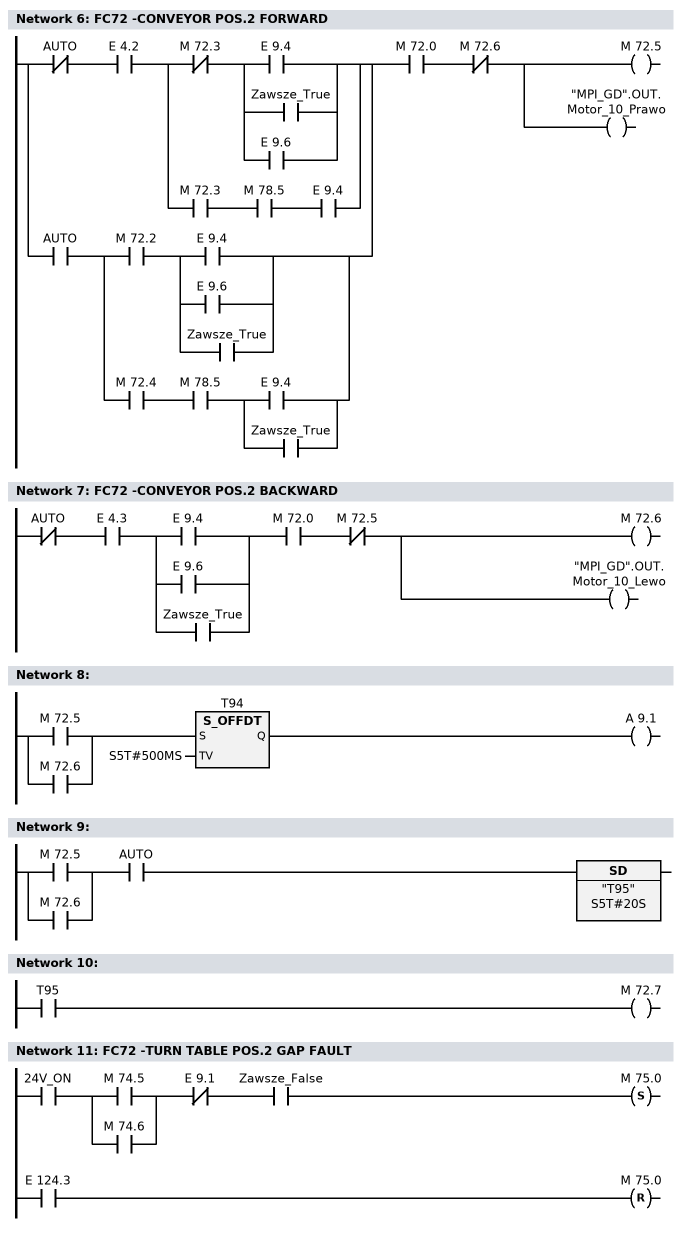
[picture p72: CONV_2 networks 6-11]
NETWORK
TITLE = FC72 -CONVEYOR POS.2 FORWARD
//Q8.2. Przenosnik jedzie do przodu
      A(;
      AN    "AUTO";
      A     "E 4.2";
      A(;
      AN    "M 72.3";
      A(;
      O     "E 9.4";
      O     "Zawsze_True";
      O     "E 9.6";
      );
      O;
      A     "M 72.3";
      A     "M 78.5";
      A     "E 9.4";
      );
      O;
      A     "AUTO";
      A(;
      A     "M 72.2";
      A(;
      O     "E 9.4";
      O     "E 9.6";
      O     "Zawsze_True";
      );
      O;
      A     "M 72.4";
      A     "M 78.5";
      A(;
      O     "E 9.4";
      O     "Zawsze_True";
      );
      );
      );
      A     "M 72.0";
      AN    "M 72.6";
      =     "M 72.5";
      =     "MPI_GD".OUT.Motor_10_Prawo;
NETWORK
TITLE = FC72 -CONVEYOR POS.2 BACKWARD
//Q8.3 przenosnik jedzie do tylu
      AN    "AUTO";
      A     "E 4.3";
      A(;
      O     "E 9.4";
      O     "E 9.6";
      O     "Zawsze_True";
      );
      A     "M 72.0";
      AN    "M 72.5";
      =     "M 72.6";
      =     "MPI_GD".OUT.Motor_10_Lewo;
NETWORK
TITLE =
      A(;
      O     "M 72.5";
      O     "M 72.6";
      );
      L     S5T#500MS;
      SF    "T94";
      NOP   0;
      NOP   0;
      NOP   0;
      A     "T94";
      =     "A 9.1";
NETWORK
TITLE =
      A(;
      O     "M 72.5";
      O     "M 72.6";
      );
      A     "AUTO";
      L     S5T#20S;
      SD    "T95";
NETWORK
TITLE =
      A     "T95";
      =     "M 72.7";
NETWORK
TITLE = FC72 -TURN TABLE POS.2 GAP FAULT
//Zablokowane
      A     "24V_ON";
      A(;
      O     "M 74.5";
      O     "M 74.6";
      );
      AN    "E 9.1";
      A     "Zawsze_False";
      S     "M 75.0";
      A     "E 124.3";
      R     "M 75.0";
      NOP   0;
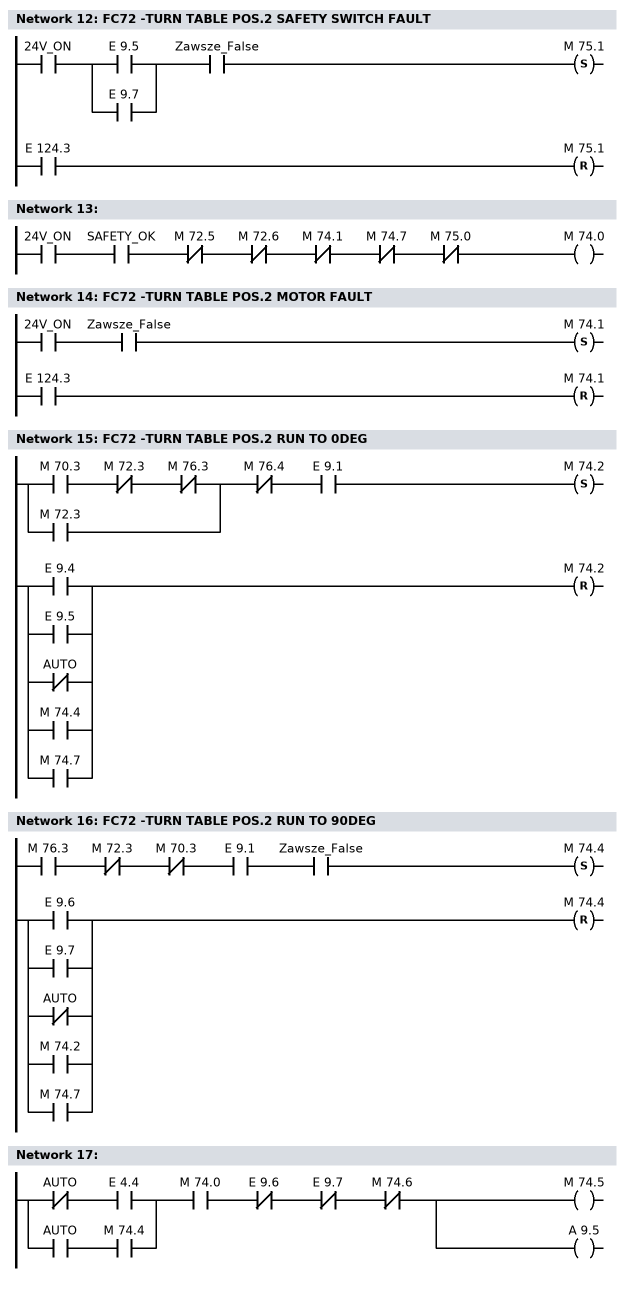
NETWORK
TITLE = FC72 -TURN TABLE POS.2 SAFETY SWITCH FAULT
//Zablokowane
      A     "24V_ON";
      A(;
      O     "E 9.5";
      O     "E 9.7";
      );
      A     "Zawsze_False";
      S     "M 75.1";
      A     "E 124.3";
      R     "M 75.1";
      NOP   0;
NETWORK
TITLE =
      A     "24V_ON";
      A     "SAFETY_OK";
      AN    "M 72.5";
      AN    "M 72.6";
      AN    "M 74.1";
      AN    "M 74.7";
      AN    "M 75.0";
      =     "M 74.0";
NETWORK
TITLE = FC72 -TURN TABLE POS.2 MOTOR FAULT
//Zablokowane.Silnik obrotnica
      A     "24V_ON";
      A     "Zawsze_False";
      S     "M 74.1";
      A     "E 124.3";
      R     "M 74.1";
      NOP   0;
NETWORK
TITLE = FC72 -TURN TABLE POS.2 RUN TO 0DEG
      A(;
      A     "M 70.3";
      AN    "M 72.3";
      AN    "M 76.3";
      O     "M 72.3";
      );
      AN    "M 76.4";
      A     "E 9.1";
      S     "M 74.2";
      A(;
      O     "E 9.4";
      O     "E 9.5";
      ON    "AUTO";
      O     "M 74.4";
      O     "M 74.7";
      );
      R     "M 74.2";
      NOP   0;
NETWORK
TITLE = FC72 -TURN TABLE POS.2 RUN TO 90DEG
//Zablokowane
      A     "M 76.3";
      AN    "M 72.3";
      AN    "M 70.3";
      A     "E 9.1";
      A     "Zawsze_False";
      S     "M 74.4";
      A(;
      O     "E 9.6";
      O     "E 9.7";
      ON    "AUTO";
      O     "M 74.2";
      O     "M 74.7";
      );
      R     "M 74.4";
      NOP   0;
NETWORK
TITLE =
      A(;
      AN    "AUTO";
      A     "E 4.4";
      O;
      A     "AUTO";
      A     "M 74.4";
      );
      A     "M 74.0";
      AN    "E 9.6";
      AN    "E 9.7";
      AN    "M 74.6";
      =     "M 74.5";
      =     "A 9.5";
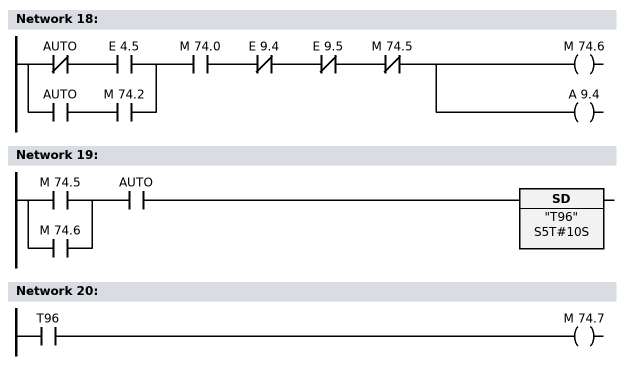
NETWORK
TITLE =
      A(;
      AN    "AUTO";
      A     "E 4.5";
      O;
      A     "AUTO";
      A     "M 74.2";
      );
      A     "M 74.0";
      AN    "E 9.4";
      AN    "E 9.5";
      AN    "M 74.5";
      =     "M 74.6";
      =     "A 9.4";
NETWORK
TITLE =
      A(;
      O     "M 74.5";
      O     "M 74.6";
      );
      A     "AUTO";
      L     S5T#10S;
      SD    "T96";
NETWORK
TITLE =
      A     "T96";
      =     "M 74.7";
END_FUNCTION

FUNCTION "Komunikacja_GD" : VOID	// FC 100
VERSION : 0.1
BEGIN
NETWORK
TITLE =
//Ten network celowo jest wolny
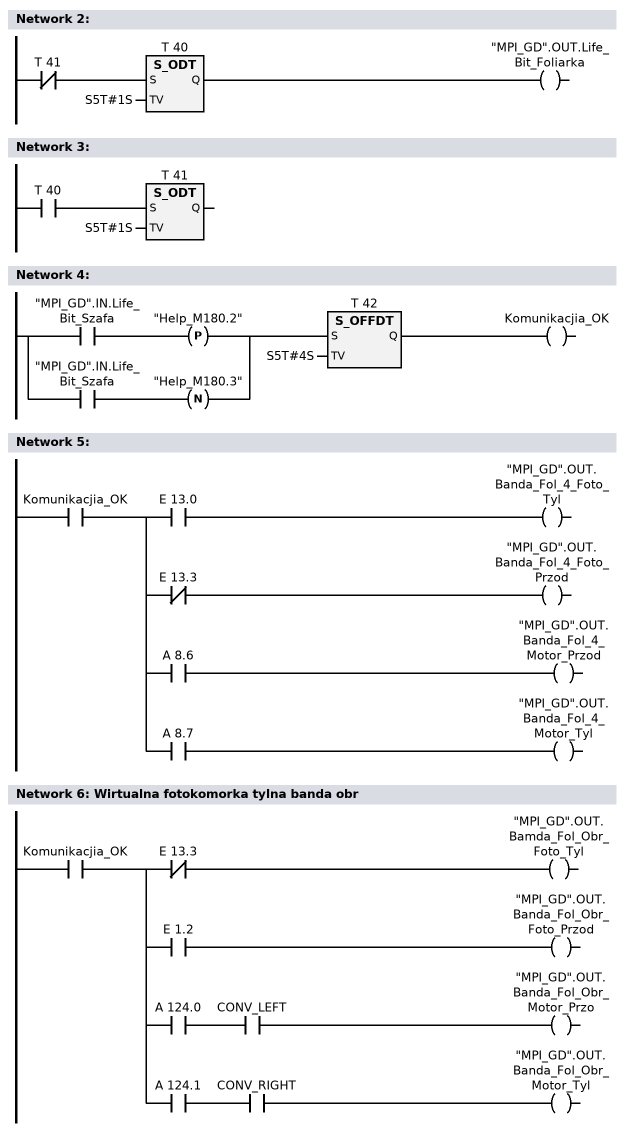
NETWORK
TITLE =
//Generator bit zycia foliarki
      AN    T 41;
      L     S5T#1S;
      SD    T 40;
      NOP   0;
      NOP   0;
      NOP   0;
      A     T 40;
      =     "MPI_GD".OUT.Life_Bit_Foliarka;
NETWORK
TITLE =
//Generator bit zycia foliarki
      A     T 40;
      L     S5T#1S;
      SD    T 41;
      NOP   0;
      NOP   0;
      NOP   0;
      NOP   0;
NETWORK
TITLE =
//Sprawdzenie komunikacji z szafa transportera
      A(;
      A     "MPI_GD".IN.Life_Bit_Szafa;
      FP    "Help_M180.2";
      O(;
      A     "MPI_GD".IN.Life_Bit_Szafa;
      FN    "Help_M180.3";
      );
      );
      L     S5T#4S;
      SF    T 42;
      NOP   0;
      NOP   0;
      NOP   0;
      A     T 42;
      =     "Komunikacjia_OK";
NETWORK
TITLE =
//Przypisanie fotokomorek do interfejsu z linia
//Jako fotokomorki tylne brane foto z muting'u
      A     "Komunikacjia_OK";
      =     L 0.0;
      A     L 0.0;
      A     "E 13.0";
      =     "MPI_GD".OUT.Banda_Fol_4_Foto_Tyl;
      A     L 0.0;
      AN    "E 13.3";
      =     "MPI_GD".OUT.Banda_Fol_4_Foto_Przod;
      A     L 0.0;
      A     "A 8.6";
      =     "MPI_GD".OUT.Banda_Fol_4_Motor_Przod;
      A     L 0.0;
      A     "A 8.7";
      =     "MPI_GD".OUT.Banda_Fol_4_Motor_Tyl;
NETWORK
TITLE = Wirtualna fotokomorka tylna banda obr
//Banda obrotowa
      A     "Komunikacjia_OK";
      =     L 0.0;
      A     L 0.0;
      AN    "E 13.3";
      =     "MPI_GD".OUT.Bamda_Fol_Obr_Foto_Tyl;
      A     L 0.0;
      A     "E 1.2";
      =     "MPI_GD".OUT.Banda_Fol_Obr_Foto_Przod;
      A     L 0.0;
      A     "A 124.0";
      A     "CONV_LEFT";
      =     "MPI_GD".OUT.Banda_Fol_Obr_Motor_Przo;
      A     L 0.0;
      A     "A 124.1";
      A     "CONV_RIGHT";
      =     "MPI_GD".OUT.Banda_Fol_Obr_Motor_Tyl;
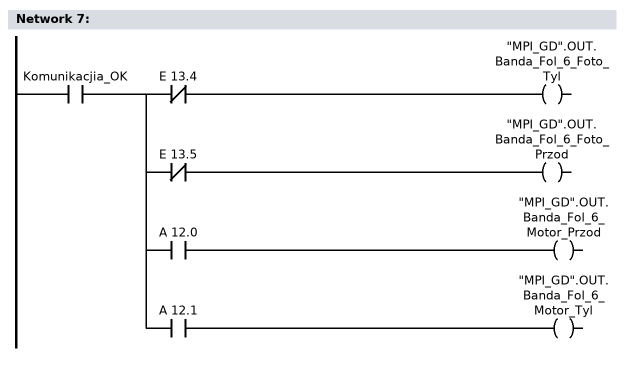
NETWORK
TITLE =
//Banda 6 jazda przod tyl
      A     "Komunikacjia_OK";
      =     L 0.0;
      A     L 0.0;
      AN    "E 13.4";
      =     "MPI_GD".OUT.Banda_Fol_6_Foto_Tyl;
      A     L 0.0;
      AN    "E 13.5";
      =     "MPI_GD".OUT.Banda_Fol_6_Foto_Przod;
      A     L 0.0;
      A     "A 12.0";
      =     "MPI_GD".OUT.Banda_Fol_6_Motor_Przod;
      A     L 0.0;
      A     "A 12.1";
      =     "MPI_GD".OUT.Banda_Fol_6_Motor_Tyl;
END_FUNCTION

FUNCTION "DISPLAY_HANDLING" : VOID	// FC 110
TITLE = HANDLING OF DATALIST PROGRAMME PARAMETERS
//DB12(RUNNING_PROG): Used in programme, copy from DB21-29 
//DB13(EDITING_PROG): New data copy to DB21-29
//DB21-29(PROG DATA): Keeping data to programme 1-9
//
//MAX 9 different programme
//MAX 24 different data to every programme
AUTHOR : LKA
NAME : DISPLAY
VERSION : 0.1
BEGIN
NETWORK
TITLE = MOVE DATA
//FLYTTA DATA
//PEKAREN ANVÄNDS FÖR ATT VÄLJA DATA I DB21 TILL 29(LISTA) DÄR DATA FÖR 
//PROGRAM (1-9) LAGRAS.
      L     "RUNNING_PROG".PRG_POINTER;
      L     20;
      +I;
      T     LW 0;
      L     21;
      >=I;
      JC    M011;
      T     LW 0;
M011: L     LW 0;
      L     29;
      <=I;
      JC    M012;
      T     LW 0;
M012: L     "RUNNING_PROG".OLD_PRG_POINTER;
      L     "RUNNING_PROG".PRG_POINTER;
      ==I;
      JC    M013;
      T     "RUNNING_PROG".OLD_PRG_POINTER;
      L     16;
      T     LW 10;
M014: L     LW 10;
      SLW   3;
      T     LD 14;
      OPN   DB [LW 0];
      L     DBW [LD 14];
      OPN   "EDITING_PROG";
      T     DBW [LD 14];
      L     LW 10;
      +     2;
      T     LW 10;
      L     54;
      <=I;
      JC    M014;
M013: L     16;
      T     LW 10;
      L     "RUNNING_PROG".PRG_POINTER;
      L     20;
      +I;
      T     LW 0;
      L     21;
      >=I;
      JC    M018;
      T     LW 0;
M018: L     LW 0;
      L     29;
      <=I;
      JC    M019;
      T     LW 0;
M019: L     LW 10;
      SLW   3;
      T     LD 14;
      OPN   "EDITING_PROG";
      L     DBW [LD 14];
      OPN   DB [LW 0];
      T     DBW [LD 14];
      L     LW 10;
      +     2;
      T     LW 10;
      L     54;
      <=I;
      JC    M019;
      L     16;
      T     LW 10;
      L     "RUNNING_PROG".PRG_CHOICE_OP3;
      L     20;
      +I;
      T     LW 0;
      L     21;
      >=I;
      JC    M016;
      T     LW 0;
M016: L     LW 0;
      L     29;
      <=I;
      JC    M017;
      T     LW 0;
M017: AN    "PULSE_PROG_REGISTER";
      AN    "PULSE_RESET";
      JC    M015;
M020: L     LW 10;
      SLW   3;
      T     LD 14;
      OPN   DB [LW 0];
      L     DBW [LD 14];
      OPN   "RUNNING_PROG";
      T     DBW [LD 14];
      L     LW 10;
      +     2;
      T     LW 10;
      L     54;
      <=I;
      JC    M020;
//TURNTABLE SPEED MIDDEL TO LOW, 90 DEGREE
      L     "RUNNING_PROG".SET_POINT_MS_TO_LS_TT;
      L     24;
      -I;
      T     "RUNNING_PROG".TT_SYNC_M_TO_L_90;
//    VÄRDE TOPPVARV
      L     "RUNNING_PROG".SET_POINT_TOPWRAP;
      L     100;
      *I;
      T     "RUNNING_PROG".TW_USED;
//    VÄRDE BOTTENVARV
      L     "RUNNING_PROG".SET_POINT_BOTTOMWRAP;
      L     100;
      *I;
      T     "RUNNING_PROG".BW_USED;
M015: NOP   0;
END_FUNCTION

FUNCTION "MANUAL_MODE" : VOID	// FC 111
TITLE = MANUAL MODE
AUTHOR : LKA
NAME : MAN_MODE
VERSION : 0.2
BEGIN
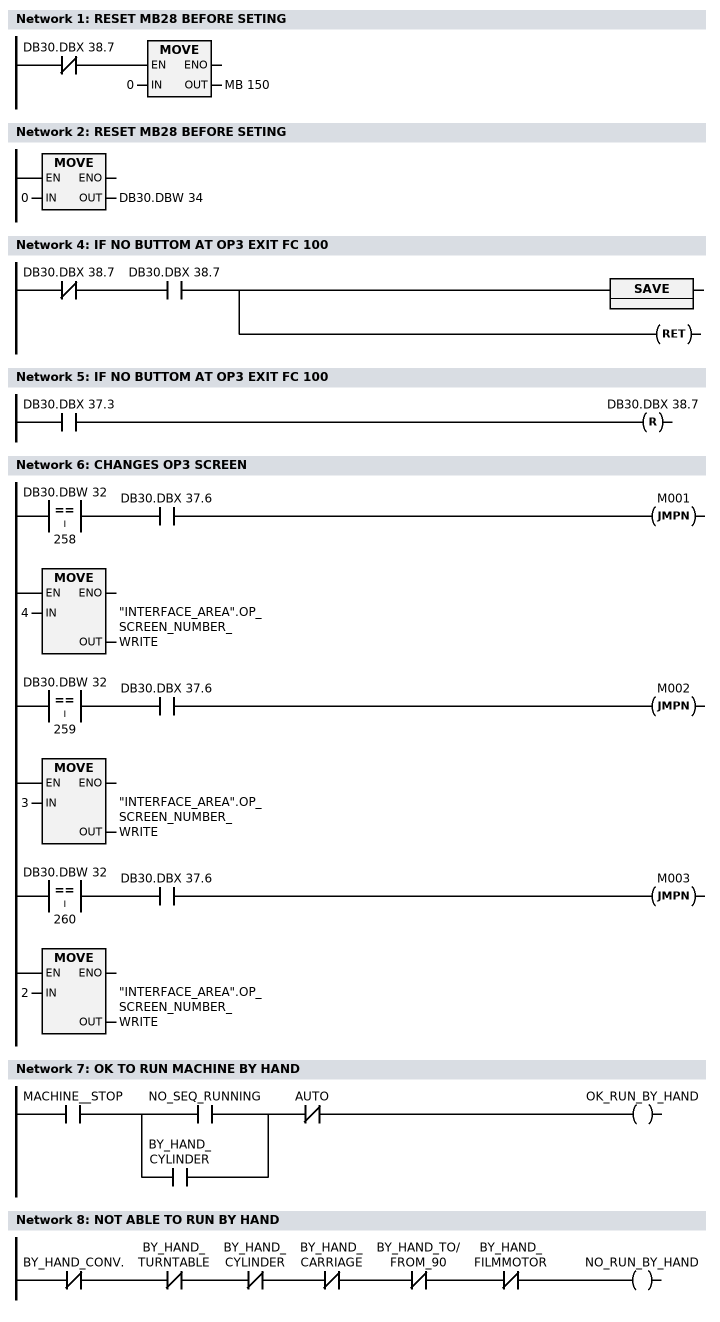
NETWORK
TITLE = RESET MB28 BEFORE SETING
      AN    DB30.DBX 38.7;
      JNB   _003;
      L     0;
      T     MB 150;
_003: NOP   0;
NETWORK
TITLE = RESET MB28 BEFORE SETING
      L     0;
      T     DB30.DBW 34;
      NOP   0;
NETWORK
TITLE = BYTA BILD I OP3, FÖRSTA TILL PROGRAMVAL.
      AN    "SUMALARM_A";
      AN    "SUMALARM_B";
      AN    "MESSAGE_SHOWING";
      JNB   OP3;
      L     DB30.DBW 32;
      L     -1;
      ==I;
      JCN   OP3;
      L     1;
      T     "INTERFACE_AREA".OP_SCREEN_NUMBER_WRITE;
OP3:  NOP   0;
NETWORK
TITLE = IF NO BUTTOM AT OP3 EXIT FC 100
      AN    DB30.DBX 38.7;
      A     DB30.DBX 38.7;
      SAVE;
      BEC;
NETWORK
TITLE = IF NO BUTTOM AT OP3 EXIT FC 100
      A     DB30.DBX 37.3;
      R     DB30.DBX 38.7;
NETWORK
TITLE = CHANGES OP3 SCREEN
//    CHANGES OP3 SCREEN TO "FILMPARAMETERS"
      L     DB30.DBW 32;
      L     258;
      ==I;
      A     DB30.DBX 37.6;
      JCN   M001;
      L     4;
      T     "INTERFACE_AREA".OP_SCREEN_NUMBER_WRITE;
M001: NOP   0;
//    CHANGES OP3 SCREEN TO "RUN MASCHINE MANUAL"
      L     DB30.DBW 32;
      L     259;
      ==I;
      A     DB30.DBX 37.6;
      JCN   M002;
      L     3;
      T     "INTERFACE_AREA".OP_SCREEN_NUMBER_WRITE;
M002: NOP   0;
//    CHANGES OP3 SCREEN TO "INFORMATION"
      L     DB30.DBW 32;
      L     260;
      ==I;
      A     DB30.DBX 37.6;
      JCN   M003;
      L     2;
      T     "INTERFACE_AREA".OP_SCREEN_NUMBER_WRITE;
M003: NOP   0;
NETWORK
TITLE = OK TO RUN MACHINE BY HAND
      A     "MACHINE__STOP";
      A(;
      O     "NO_SEQ_RUNNING";
      O     "BY_HAND_CYLINDER";
      );
      AN    "AUTO";
      =     "OK_RUN_BY_HAND";
NETWORK
TITLE = NOT ABLE TO RUN BY HAND
      AN    "BY_HAND_CONV.";
      AN    "BY_HAND_TURNTABLE";
      AN    "BY_HAND_CYLINDER";
      AN    "BY_HAND_CARRIAGE";
      AN    "BY_HAND_TO/FROM_90";
      AN    "BY_HAND_FILMMOTOR";
      =     "NO_RUN_BY_HAND";
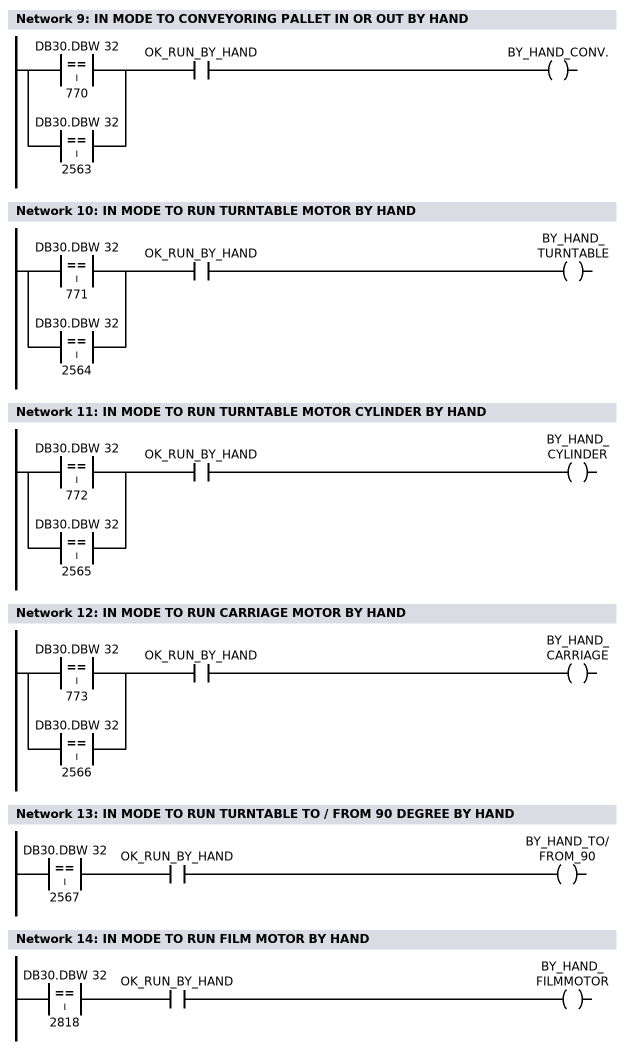
NETWORK
TITLE = IN MODE TO CONVEYORING PALLET IN OR OUT BY HAND
      A(;
      O(;
      L     DB30.DBW 32;
      L     770;
      ==I;
      );
      O(;
      L     DB30.DBW 32;
      L     2563;
      ==I;
      );
      );
      A     "OK_RUN_BY_HAND";
      =     "BY_HAND_CONV.";
NETWORK
TITLE = IN MODE TO RUN TURNTABLE MOTOR BY HAND
      A(;
      O(;
      L     DB30.DBW 32;
      L     771;
      ==I;
      );
      O(;
      L     DB30.DBW 32;
      L     2564;
      ==I;
      );
      );
      A     "OK_RUN_BY_HAND";
      =     "BY_HAND_TURNTABLE";
NETWORK
TITLE = IN MODE TO RUN TURNTABLE MOTOR CYLINDER BY HAND
      A(;
      O(;
      L     DB30.DBW 32;
      L     772;
      ==I;
      );
      O(;
      L     DB30.DBW 32;
      L     2565;
      ==I;
      );
      );
      A     "OK_RUN_BY_HAND";
      =     "BY_HAND_CYLINDER";
NETWORK
TITLE = IN MODE TO RUN CARRIAGE MOTOR BY HAND
      A(;
      O(;
      L     DB30.DBW 32;
      L     773;
      ==I;
      );
      O(;
      L     DB30.DBW 32;
      L     2566;
      ==I;
      );
      );
      A     "OK_RUN_BY_HAND";
      =     "BY_HAND_CARRIAGE";
NETWORK
TITLE = IN MODE TO RUN TURNTABLE TO / FROM 90 DEGREE BY HAND
      A(;
      L     DB30.DBW 32;
      L     2567;
      ==I;
      );
      A     "OK_RUN_BY_HAND";
      =     "BY_HAND_TO/FROM_90";
NETWORK
TITLE = IN MODE TO RUN FILM MOTOR BY HAND
      A(;
      L     DB30.DBW 32;
      L     2818;
      ==I;
      );
      A     "OK_RUN_BY_HAND";
      =     "BY_HAND_FILMMOTOR";
END_FUNCTION

FUNCTION "ALARM" : VOID	// FC 120
TITLE = ALARM
AUTHOR : LKA
NAME : ALARM
VERSION : 0.1
BEGIN
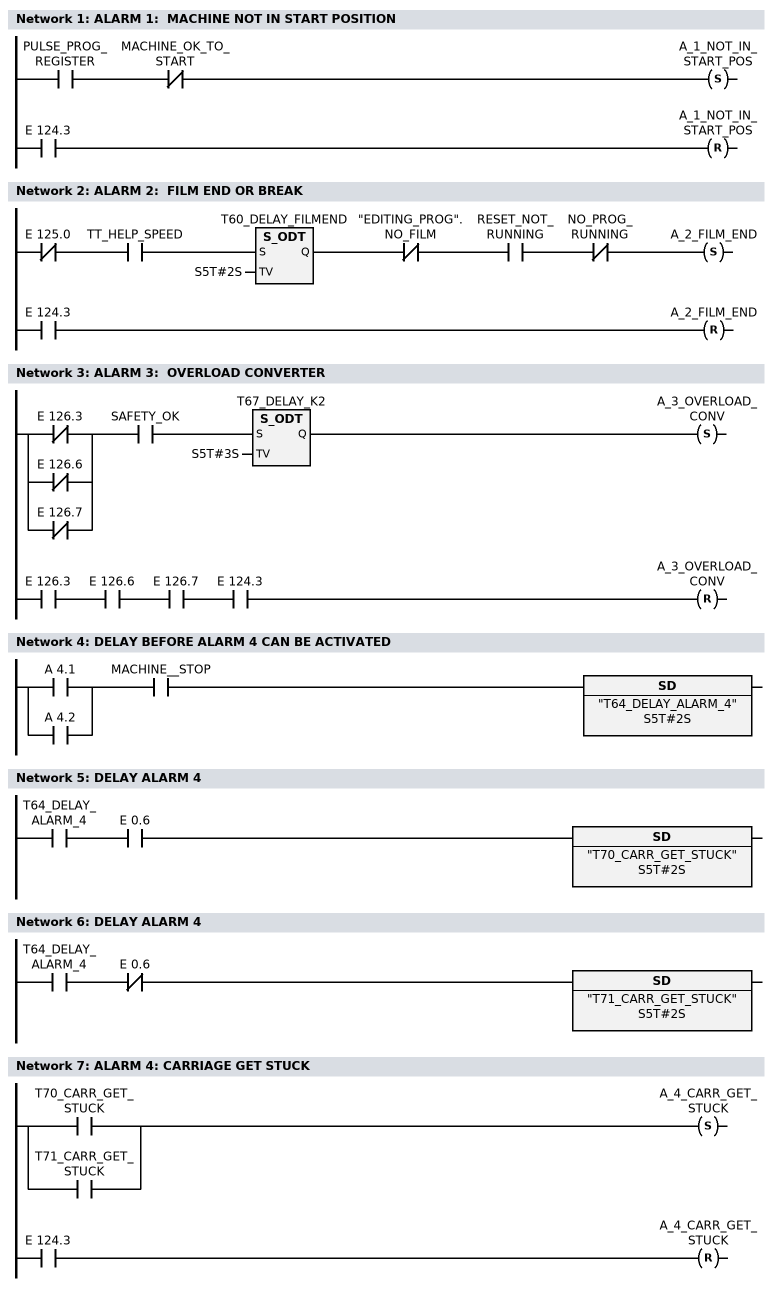
NETWORK
TITLE = ALARM 1:  MACHINE NOT IN START POSITION
//LARM EJ UTGÅNGSLÄGE
      A     "PULSE_PROG_REGISTER";
      AN    "MACHINE_OK_TO_START";
      S     "A_1_NOT_IN_START_POS";
      A     "E 124.3";
      R     "A_1_NOT_IN_START_POS";
      NOP   0;
NETWORK
TITLE = ALARM 2:  FILM END OR BREAK
//LARM SLUT FILM/FILMBROTT
      A(;
      AN    "E 125.0";
      A     "TT_HELP_SPEED";
      L     S5T#2S;
      SD    "T60_DELAY_FILMEND";
      NOP   0;
      NOP   0;
      NOP   0;
      A     "T60_DELAY_FILMEND";
      );
      AN    "EDITING_PROG".NO_FILM;
      A     "RESET_NOT_RUNNING";
      AN    "NO_PROG_RUNNING";
      S     "A_2_FILM_END";
      A     "E 124.3";
      R     "A_2_FILM_END";
      NOP   0;
NETWORK
TITLE = ALARM 3:  OVERLOAD CONVERTER
//LARM ÖVERBELASTNING OMRIKTARE
      AN    "E 126.3";
      ON    "E 126.6";
      ON    "E 126.7";
      A(;
      A     "SAFETY_OK";
      L     S5T#3S;
      SD    "T67_DELAY_K2";
      NOP   0;
      NOP   0;
      NOP   0;
      A     "T67_DELAY_K2";
      );
      S     "A_3_OVERLOAD_CONV";
      A     "E 126.3";
      A     "E 126.6";
      A     "E 126.7";
      A     "E 124.3";
      R     "A_3_OVERLOAD_CONV";
      NOP   0;
NETWORK
TITLE = DELAY BEFORE ALARM 4 CAN BE ACTIVATED
      A(;
      O     "A 4.1";
      O     "A 4.2";
      );
      A     "MACHINE__STOP";
      L     S5T#2S;
      SD    "T64_DELAY_ALARM_4";
NETWORK
TITLE = DELAY ALARM 4
      A     "T64_DELAY_ALARM_4";
      A     "E 0.6";
      L     S5T#2S;
      SD    "T70_CARR_GET_STUCK";
NETWORK
TITLE = DELAY ALARM 4
      A     "T64_DELAY_ALARM_4";
      AN    "E 0.6";
      L     S5T#2S;
      SD    "T71_CARR_GET_STUCK";
NETWORK
TITLE = ALARM 4: CARRIAGE GET STUCK
//LARM HISSEN HAR FASTNAT
      A(;
      O     "T70_CARR_GET_STUCK";
      O     "T71_CARR_GET_STUCK";
      );
      S     "A_4_CARR_GET_STUCK";
      A     "E 124.3";
      R     "A_4_CARR_GET_STUCK";
      NOP   0;
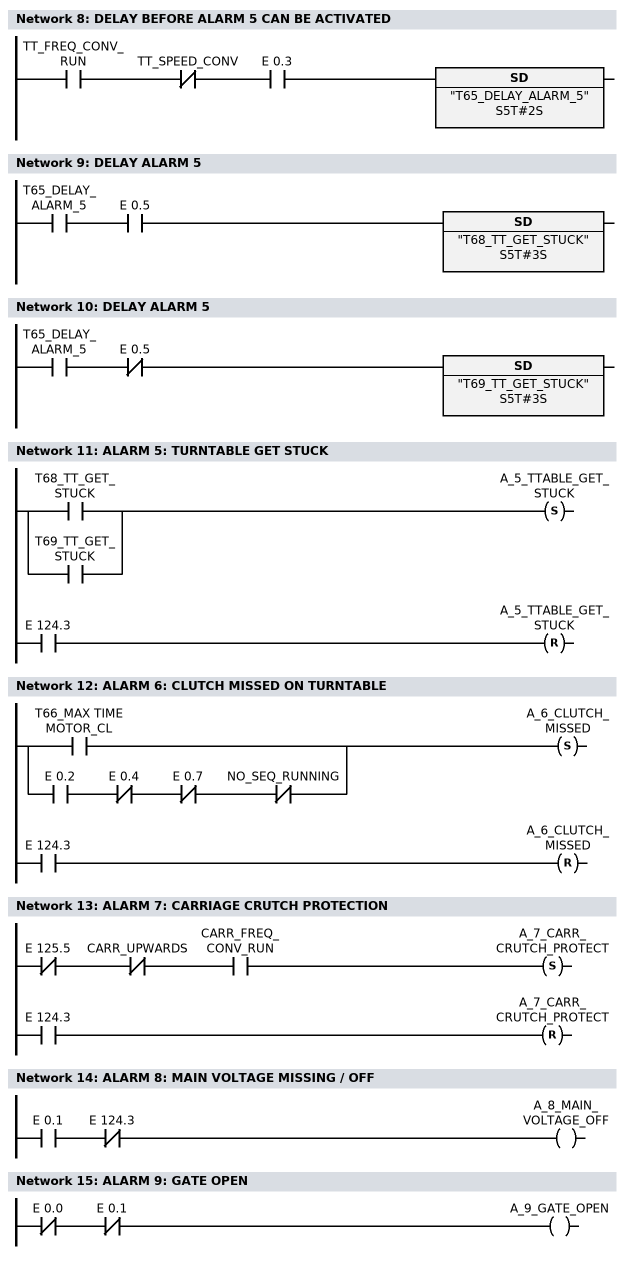
NETWORK
TITLE = DELAY BEFORE ALARM 5 CAN BE ACTIVATED
      A     "TT_FREQ_CONV_RUN";
      AN    "TT_SPEED_CONV";
      A     "E 0.3";
      L     S5T#2S;
      SD    "T65_DELAY_ALARM_5";
NETWORK
TITLE = DELAY ALARM 5
      A     "T65_DELAY_ALARM_5";
      A     "E 0.5";
      L     S5T#3S;
      SD    "T68_TT_GET_STUCK";
NETWORK
TITLE = DELAY ALARM 5
      A     "T65_DELAY_ALARM_5";
      AN    "E 0.5";
      L     S5T#3S;
      SD    "T69_TT_GET_STUCK";
NETWORK
TITLE = ALARM 5: TURNTABLE GET STUCK
//LARM BORDET HAR FASTNAT
      A(;
      O     "T68_TT_GET_STUCK";
      O     "T69_TT_GET_STUCK";
      );
      S     "A_5_TTABLE_GET_STUCK";
      A     "E 124.3";
      R     "A_5_TTABLE_GET_STUCK";
      NOP   0;
NETWORK
TITLE = ALARM 6: CLUTCH MISSED ON TURNTABLE
//LARM MISSAT KOPPLING
      A(;
      O     "T66_MAX TIME MOTOR_CL";
      O;
      A     "E 0.2";
      AN    "E 0.4";
      AN    "E 0.7";
      AN    "NO_SEQ_RUNNING";
      );
      S     "A_6_CLUTCH_MISSED";
      A     "E 124.3";
      R     "A_6_CLUTCH_MISSED";
      NOP   0;
NETWORK
TITLE = ALARM 7: CARRIAGE CRUTCH PROTECTION
//LARM KLÄMMSKYDD HISS
      AN    "E 125.5";
      AN    "CARR_UPWARDS";
      A     "CARR_FREQ_CONV_RUN";
      S     "A_7_CARR_CRUTCH_PROTECT";
      A     "E 124.3";
      R     "A_7_CARR_CRUTCH_PROTECT";
      NOP   0;
NETWORK
TITLE = ALARM 8: MAIN VOLTAGE MISSING / OFF
//LARM MASKINSTOPP AKTIVERAT
      A     "E 0.1";
      AN    "E 124.3";
      =     "A_8_MAIN_VOLTAGE_OFF";
NETWORK
TITLE = ALARM 9: GATE OPEN
//LARM NÖDSTOPP AKTIVERAT
      AN    "E 0.0";
      AN    "E 0.1";
      =     "A_9_GATE_OPEN";
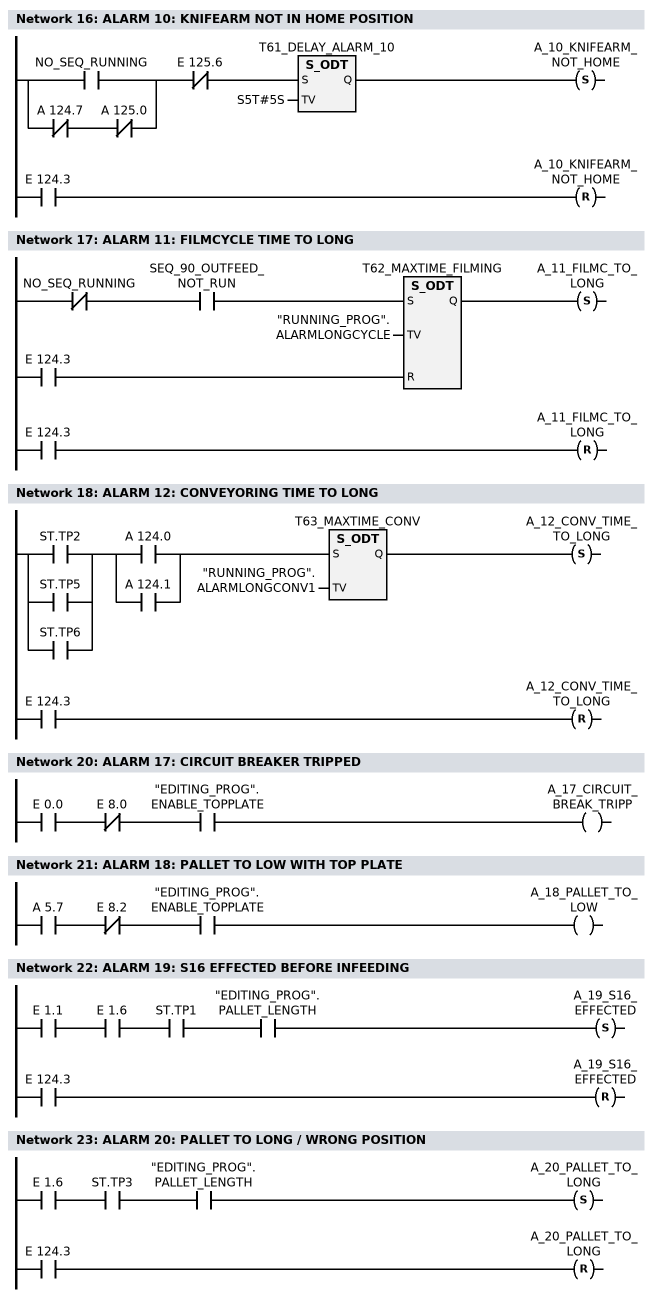
NETWORK
TITLE = ALARM 10: KNIFEARM NOT IN HOME POSITION
      A(;
      A(;
      O     "NO_SEQ_RUNNING";
      O;
      AN    "A 124.7";
      AN    "A 125.0";
      );
      AN    "E 125.6";
      L     S5T#5S;
      SD    "T61_DELAY_ALARM_10";
      NOP   0;
      NOP   0;
      NOP   0;
      A     "T61_DELAY_ALARM_10";
      );
      S     "A_10_KNIFEARM_NOT_HOME";
      A     "E 124.3";
      R     "A_10_KNIFEARM_NOT_HOME";
      NOP   0;
NETWORK
TITLE = ALARM 11: FILMCYCLE TIME TO LONG
//LARM FILMTID LÅNG
      A(;
      AN    "NO_SEQ_RUNNING";
      A     "SEQ_90_OUTFEED_NOT_RUN";
      L     "RUNNING_PROG".ALARMLONGCYCLE;
      SD    "T62_MAXTIME_FILMING";
      A     "E 124.3";
      R     "T62_MAXTIME_FILMING";
      NOP   0;
      NOP   0;
      A     "T62_MAXTIME_FILMING";
      );
      S     "A_11_FILMC_TO_LONG";
      A     "E 124.3";
      R     "A_11_FILMC_TO_LONG";
      NOP   0;
NETWORK
TITLE = ALARM 12: CONVEYORING TIME TO LONG
//LARM TRANSPORTTID FÖR LÅNG
      A(;
      A(;
      O     "ST.TP2";
      O     "ST.TP5";
      O     "ST.TP6";
      );
      A(;
      O     "A 124.0";
      O     "A 124.1";
      );
      L     "RUNNING_PROG".ALARMLONGCONV1;
      SD    "T63_MAXTIME_CONV";
      NOP   0;
      NOP   0;
      NOP   0;
      A     "T63_MAXTIME_CONV";
      );
      S     "A_12_CONV_TIME_TO_LONG";
      A     "E 124.3";
      R     "A_12_CONV_TIME_TO_LONG";
      NOP   0;
NETWORK
TITLE = ALARM 13: PALLET PAUSED DURING CONVEYORING IN TO MACHINE
//LARM TRANSPORTTID FÖR LÅNG
      A(;
      A     "ST.TP2";
      A     "E 1.2";
      AN    "A 124.0";
      AN    "A 124.1";
      S     M 249.1;
      A     "A_13_PALLET_PAUSED";
      R     M 249.1;
      A     M 249.1;
      );
      AN    "ST.TP2";
      S     "A_13_PALLET_PAUSED";
      A     "E 124.3";
      R     "A_13_PALLET_PAUSED";
      NOP   0;
NETWORK
TITLE = ALARM 17: CIRCUIT BREAKER TRIPPED
//LARM AUTOMATSÄKRING UTLÖST
      A     "E 0.0";
      AN    "E 8.0";
      A     "EDITING_PROG".ENABLE_TOPPLATE;
      =     "A_17_CIRCUIT_BREAK_TRIPP";
NETWORK
TITLE = ALARM 18: PALLET TO LOW WITH TOP PLATE
//PALL FÖR LÅG MED TOPPLATTA
      A     "A 5.7";
      AN    "E 8.2";
      A     "EDITING_PROG".ENABLE_TOPPLATE;
      =     "A_18_PALLET_TO_LOW";
NETWORK
TITLE = ALARM 19: S16 EFFECTED BEFORE INFEEDING
//LARM AUTOMATSÄKRING UTLÖST
      A     "E 1.1";
      A     "E 1.6";
      A     "ST.TP1";
      A     "EDITING_PROG".PALLET_LENGTH;
      S     "A_19_S16_EFFECTED";
      A     "E 124.3";
      R     "A_19_S16_EFFECTED";
      NOP   0;
NETWORK
TITLE = ALARM 20: PALLET TO LONG / WRONG POSITION
//LARM AUTOMATSÄKRING UTLÖST
      A     "E 1.6";
      A     "ST.TP3";
      A     "EDITING_PROG".PALLET_LENGTH;
      S     "A_20_PALLET_TO_LONG";
      A     "E 124.3";
      R     "A_20_PALLET_TO_LONG";
      NOP   0;
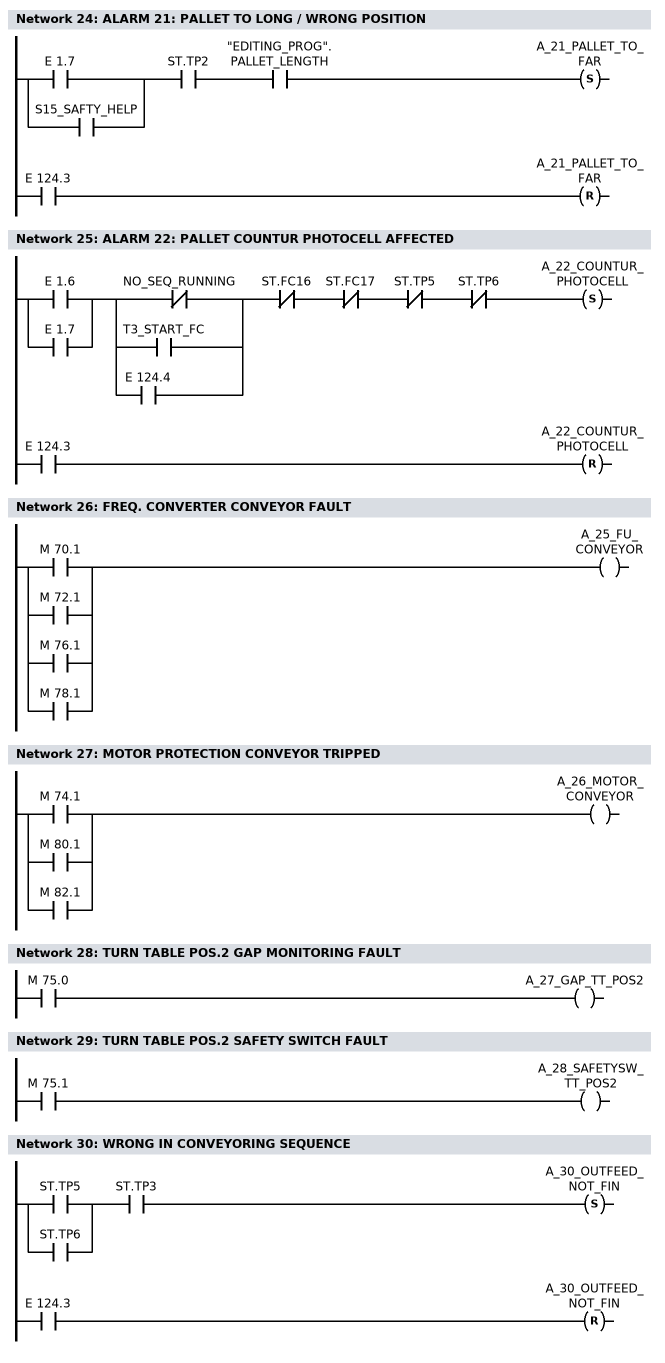
NETWORK
TITLE = ALARM 21: PALLET TO LONG / WRONG POSITION
//S15, THIRD SAFETY POTOCELL EFFECTED DURING INFEEDING, OPTION WITH 90 DEGREE.
      A(;
      O     "E 1.7";
      O     "S15_SAFTY_HELP";
      );
      A     "ST.TP2";
      A     "EDITING_PROG".PALLET_LENGTH;
      S     "A_21_PALLET_TO_FAR";
      A     "E 124.3";
      R     "A_21_PALLET_TO_FAR";
      NOP   0;
NETWORK
TITLE = ALARM 22: PALLET COUNTUR PHOTOCELL AFFECTED
//LARM 
      A(;
      O     "E 1.6";
      O     "E 1.7";
      );
      A(;
      ON    "NO_SEQ_RUNNING";
      O     "T3_START_FC";
      O     "E 124.4";
      );
      AN    "ST.FC16";
      AN    "ST.FC17";
      AN    "ST.TP5";
      AN    "ST.TP6";
      S     "A_22_COUNTUR_PHOTOCELL";
      A     "E 124.3";
      R     "A_22_COUNTUR_PHOTOCELL";
      NOP   0;
NETWORK
TITLE = FREQ. CONVERTER CONVEYOR FAULT
      O     "M 70.1";
      O     "M 72.1";
      O     "M 76.1";
      O     "M 78.1";
      =     "A_25_FU_CONVEYOR";
NETWORK
TITLE = MOTOR PROTECTION CONVEYOR TRIPPED
      O     "M 74.1";
      O     "M 80.1";
      O     "M 82.1";
      =     "A_26_MOTOR_CONVEYOR";
NETWORK
TITLE = TURN TABLE POS.2 GAP MONITORING FAULT
      A     "M 75.0";
      =     "A_27_GAP_TT_POS2";
NETWORK
TITLE = TURN TABLE POS.2 SAFETY SWITCH FAULT
      A     "M 75.1";
      =     "A_28_SAFETYSW_TT_POS2";
NETWORK
TITLE = WRONG IN CONVEYORING SEQUENCE
//OUTFEEDING NOT FINISHED THEN INFEEDING PALLET STOP.
//LARM FÖR FEL I TRANSPORTSEKVENS, UTTRANSPORT PÅGÅR FAST INTRANSPORT ÄR KLART.
      A(;
      O     "ST.TP5";
      O     "ST.TP6";
      );
      A     "ST.TP3";
      S     "A_30_OUTFEED_NOT_FIN";
      A     "E 124.3";
      R     "A_30_OUTFEED_NOT_FIN";
      NOP   0;
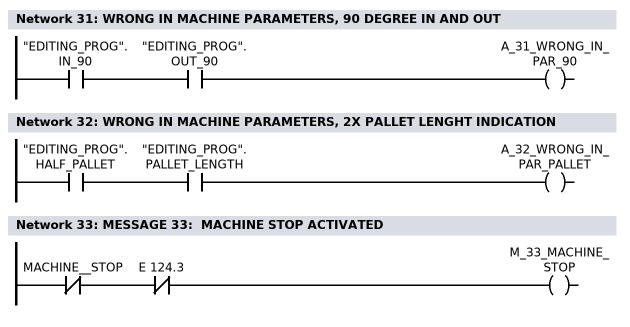
NETWORK
TITLE = WRONG IN MACHINE PARAMETERS, 90 DEGREE IN AND OUT
//LARM FÖR FEL I MASKINPARAMETRAR, VALT BÅDE 90 IN OCH 90 UT = GÅR EJ I STD VERS.
      A     "EDITING_PROG".IN_90;
      A     "EDITING_PROG".OUT_90;
      =     "A_31_WRONG_IN_PAR_90";
NETWORK
TITLE = WRONG IN MACHINE PARAMETERS, 2X PALLET LENGHT INDICATION
//LARM FÖR FEL I MASKINPARAMETRAR, VALT BÅDE 90 IN OCH 90 UT = GÅR EJ I STD VERS.
      A     "EDITING_PROG".HALF_PALLET;
      A     "EDITING_PROG".PALLET_LENGTH;
      =     "A_32_WRONG_IN_PAR_PALLET";
NETWORK
TITLE = MESSAGE 33:  MACHINE STOP ACTIVATED
//MEDDELANDE MASKINSTOPP AKTIVERAT
      AN    "MACHINE__STOP";
      AN    "E 124.3";
      =     "M_33_MACHINE_STOP";
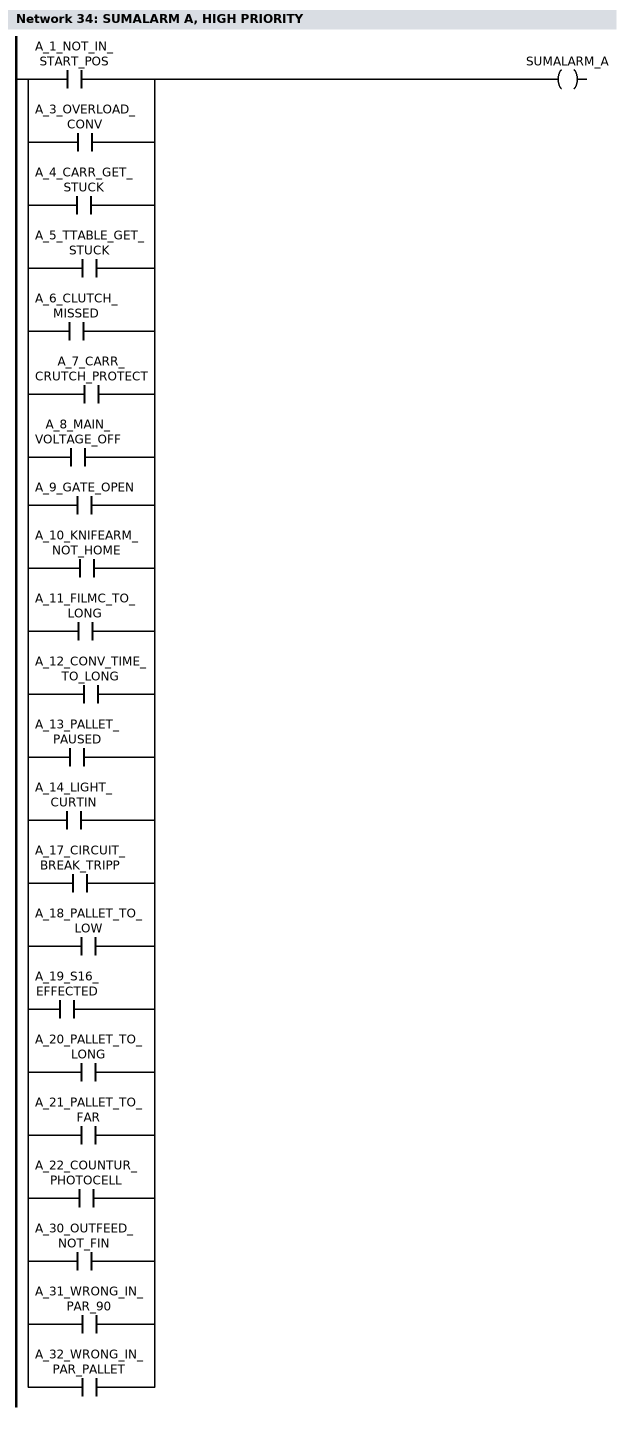
NETWORK
TITLE = SUMALARM A, HIGH PRIORITY
//SUMMALARM A, HÖG PRIORITET
//
      NOP   0;
      O     "A_1_NOT_IN_START_POS";
      O     "A_3_OVERLOAD_CONV";
      O     "A_4_CARR_GET_STUCK";
      O     "A_5_TTABLE_GET_STUCK";
      O     "A_6_CLUTCH_MISSED";
      O     "A_7_CARR_CRUTCH_PROTECT";
      O     "A_8_MAIN_VOLTAGE_OFF";
      O     "A_9_GATE_OPEN";
      O     "A_10_KNIFEARM_NOT_HOME";
      O     "A_11_FILMC_TO_LONG";
      O     "A_12_CONV_TIME_TO_LONG";
      O     "A_13_PALLET_PAUSED";
      O     "A_14_LIGHT_CURTIN";
      O     "A_17_CIRCUIT_BREAK_TRIPP";
      O     "A_18_PALLET_TO_LOW";
      O     "A_19_S16_EFFECTED";
      O     "A_20_PALLET_TO_LONG";
      O     "A_21_PALLET_TO_FAR";
      O     "A_22_COUNTUR_PHOTOCELL";
      O     "A_30_OUTFEED_NOT_FIN";
      O     "A_31_WRONG_IN_PAR_90";
      O     "A_32_WRONG_IN_PAR_PALLET";
      =     "SUMALARM_A";
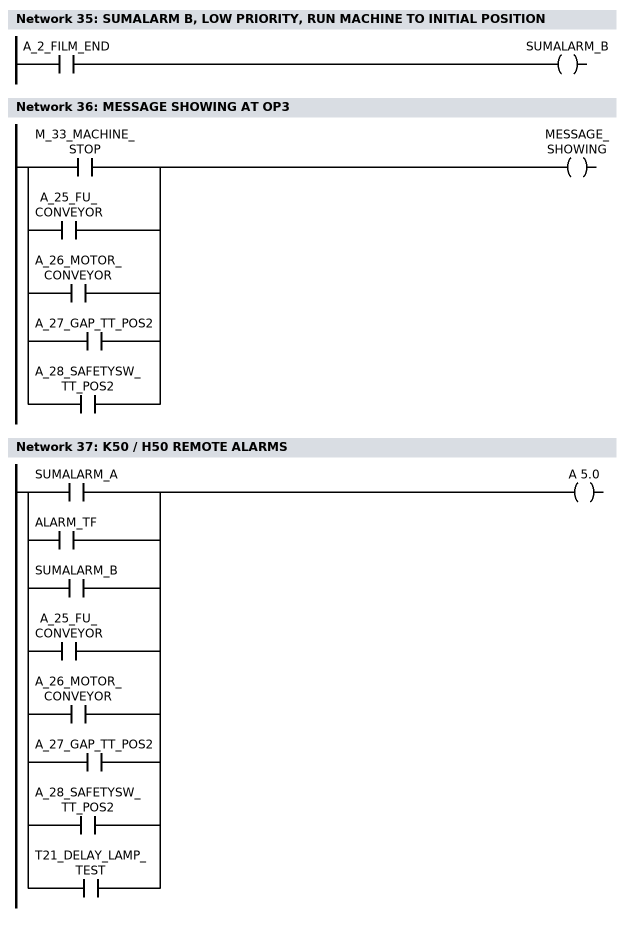
NETWORK
TITLE = SUMALARM B, LOW PRIORITY, RUN MACHINE TO INITIAL POSITION
//SUMMALARM B, LÅG PRIORITET
      A     "A_2_FILM_END";
      =     "SUMALARM_B";
NETWORK
TITLE = MESSAGE SHOWING AT OP3
      O     "M_33_MACHINE_STOP";
      O     "A_25_FU_CONVEYOR";
      O     "A_26_MOTOR_CONVEYOR";
      O     "A_27_GAP_TT_POS2";
      O     "A_28_SAFETYSW_TT_POS2";
      =     "MESSAGE_SHOWING";
NETWORK
TITLE = K50 / H50 REMOTE ALARMS
//OBS! DRAR BÅDE LAMPA OCH RELÄ
      O     "SUMALARM_A";
      O     "ALARM_TF";
      O     "SUMALARM_B";
      O     "A_25_FU_CONVEYOR";
      O     "A_26_MOTOR_CONVEYOR";
      O     "A_27_GAP_TT_POS2";
      O     "A_28_SAFETYSW_TT_POS2";
      O     "T21_DELAY_LAMP_TEST";
      =     "A 5.0";
END_FUNCTION

DATA_BLOCK "RUNNING_PROG"	// DB 12
AUTHOR : LKA
NAME : MAINDATA
VERSION : 0.1
  STRUCT
   PRG_CHOICE_OP3 : INT  := 1;	//PROGRAMME CHOICE FROM OP3
   EXTERNAL_PROGRAMME : INT ;	//EXTERNAL PROGRAMME CHOICE
   OLD_PRG_POINTER : INT ;	//OLD PROGRAMME VALUE
   PRG_POINTER : INT  := 1;	//PROGRAMME WHICH PARAMETR IS TO BE CHANGED
   ACTUAL_PROGRAMME : INT ;	//AKTUELLT PROGRAM SOM ANVÄNDS I FILMCYKELN
   ACTUAL_PROGRAMME_JUMP : INT ;	//JUMP VALUE TO FC 21-29
   SPARE_12 : INT ;
   SPARE_14 : INT ;
   FILMTENSION_TOP : INT  := 10;	//SET POINT FILMTENSION TOP
   FILMTENSION_MIDDLE : INT  := 10;	//SET POINT FILMTENSION MIDDLE
   FILMTENSION_BOTTOM : INT  := 10;	//SET POINT FILMTENSION BOTTOM
   SET_POINT_TOPWRAP : INT  := 1;	//SET POINT NUMBER OF TOPWRAP
   SET_POINT_BOTTOMWRAP : INT  := 2;	//SET POINT NUMBER OF BOTTOMWRAP
   SET_POINT_MS_TO_LS_TT : INT  := 66;	//SET POINT MEDDLE SPEED BEFORE LOW SPEED, TURNTABLE
   SET_POINT_MID_SPEED_TT : INT  := 40;	//SET POINT MEDDLE SPEED, TURNTABLE
   SET_POINT_HI_SPEED_TT : INT  := 55;	//SET POINT HIGH SPEED, TURNTABLE
   SET_POINT_WRA_SPEED_DOWN : INT  := 35;	//SET POINT WRAPPING SPEED DOWNWARDS, CARRIAGE
   SET_POINT_WRAPP_SPEED_UP : INT  := 35;	//SET POINT WRAPPING SPEED UPWARDS, CARRIAGE
   SET_POINT_HI_SPEED_CARR : INT  := 100;	//SET POINT HIGH SPEED, CARRIAGE
   TOP_PLATE : BOOL  := TRUE;	//PROGRAMME LAY OUT TOP PLATE
   TOP_FILM : BOOL ;	//PROGRAMME LAY OUT TOP FILM
   WATERPROFE_TOP_FILM : BOOL ;	//PROGRAMME LAY OUT LOADCASSETTE
   FILMWELDING : BOOL  := TRUE;	//PROGRAMME LAY OUT FILMWELDING
   HOT_AIR_FILMWELDING : BOOL ;	//PROGRAMME LAY OUT HOT AIR FILMWELDING
   SPARE_40 : INT ;
   SPARE_42 : INT ;
   SPARE_44 : INT ;
   CARR_STOP_AFTER_PC : INT  := 3;	//CARRIAGE STOP AFTER PHOTOCELL
   CARR_DOWN_BEFORE_CUT : INT ;	//CARRIAGE DOWN BEFORE CUTTING
   FILMWELDIND_TIME : S5TIME  := S5T#400MS;	//FILMWELDING TIME
   SET_POINT_CONT_BEFORE_HS : INT  := 100;	//SET POINT PULSES BEFORE HIGH SPEED
   SPARE_54 : INT ;
   SPARE_56 : INT ;
   SPARE_58 : INT ;
   TT_SYNC_M_TO_L_90 : INT ;	//MIDDLE TO LOW SPEED, 90 DEG
   CNT_TURNTABLE_FROM_START : INT ;	//COUNTER TURNTABLE POSITION FROM START
   CNT_FILMHOLDER_OUT : INT ;	//COUNTER FILMHOLDER OUT
   CNT_PULSES_ACT_WRAP : INT ;	//NUMBER OF PULSES ACTUAL WRAP, I 0.4 = 0
   CNT_TOP_WRAP : INT ;	//COUNTER TOP WRAP
   CNT_BOTTOM_WRAP : INT ;	//COUNTER BOTTOM WRAP
   OLD_TT_POS_TO_ALARM : INT ;	//OLD TURNTABLE POSITION, HELP TO ALARM 20
   RET_TURNTABLE : INT  := 95;	//TURNTABLE CONSTANT, DECELERATION
   TW_USED : INT ;	//TOP WRAP VALUE IN PULSES
   BW_USED : INT ;	//BOTTOM WRAP VALUE IN PULSES
   FILMHOLDER_HOME : INT  := 125;	//FILMHOLDER HOME
   OK_TO_SYNC_TURNTABLE : INT  := 20;	//OK TO SYNCHRONICE TURNTABLE CONSIDER CARRIAGE
   VALUE_CLUTCH_OFF : INT  := 50;	//VALUE THEN OK TO TURN CLUTCH OFF
   TT_LOW_SPEED : INT  := 6;	//SET POINT LOW SPEED, TURNTABLE
   TT_CONV_SPEED : INT  := 25;	//SET POINT CONVEYORING SPEED, TURNTABLE
   SPARE_90 : INT ;
   SPARE_92 : INT ;
   FFS_END_LEVEL : INT  := 2000;	//FILM FEED SYSTEM, END LEVEL, AFTER CLUTCH OFF
   FFS_START_LEVEL : INT  := 4000;	//FILM FEED SYSTEM, START LEVEL, VALUE FILMMOTOR
   FFS_STEPS : INT  := 100;	//VALUE TO INCREASE VALUE FILMMOTOR
   CONVEYOR_STOP_T0 : S5TIME  := S5T#3S250MS;	//DELAY TIME CONVEYOR STOP, PALLET ON MACHINE
   OUTFEEDING_TIME_T1 : S5TIME  := S5T#500MS;	//CONVEYOR OUTFEEDING TIME
   DELAY_MOTOR_TO_CLUTCH_T2 : S5TIME  := S5T#100MS;	//DELAY START MOTOR TO CLUTCH
   DELAY_FC_START_T3 : S5TIME  := S5T#100MS;	//DELAY FILM CYCLE START
   FILTER_S1254_PALLET_H_T4 : S5TIME  := S5T#300MS;	//FILTER TIME TO S1254, PALLET HIGH
   CLAMP_T5 : S5TIME  := S5T#100MS;	//DELAY TIME FILMHOLDER OPEN/TURN
   CUTTING_T6 : S5TIME  := S5T#3S;	//DELAY TIME CUTTING
   KNIFEARM_BACK_T7 : S5TIME  := S5T#2S;	//DELAY TIME CUTTING ARM 1/2 HOME
   ALARMLONGCYCLE : S5TIME  := S5T#1M30S;	//DELAY TIME ALARM LONG FILMCYCLE
   FILMHOLDER_CLOSE_T9 : S5TIME  := S5T#1S;	//DELAY TIME FILMHOLDER CLOSE
   KNIFE_UP_T10 : S5TIME  := S5T#400MS;	//DELAY TIME KNIFE UP
   CUTTING_ARM_HOME_T11 : S5TIME  := S5T#1S;	//DELAY TIME CUTTING ARM HOME
   T12_DELAY_TT_STOP_0 : S5TIME  := S5T#300MS;	//DELAY TIME STOP TURNTABLE IN 0 DEGREE
   T13_DELAY_TT_STOP_90 : S5TIME ;	//DELAY TIME STOP TURNTABLE IN 90 DEGREE (FC)
   T14_DELAY_TT_S_TO_90 : S5TIME ;	//DELAY TIME STOP TURNTABLE FROM 0 TO 90 DEGREE
   T51_T53_DELAY_TIME : S5TIME  := S5T#250MS;	//OFF DELAY TIME TO SIGNAL, LENGTH MEASURING
   T16_TIME_MS_TO_90 : S5TIME  := S5T#1S500MS;	//TIME TO RUN TURNTABLE IN MIDDLE SPEED TO/FROM 90 DEGREE
   ALARMLONGCONV1 : S5TIME  := S5T#45S;	//DELAY TIME ALARM LONG CONVEUORING
   T52_CONV_STOP_HALF_P : S5TIME ;	//DELAY TIME CONVEYOR STOP, HALF PALLET ON MACHINE, OPTION
   CNT_CARR_UP_IN_RESET : INT  := 34;	//COUNTER CARRIAGE UPWARDS IN RESET
   RET_HISS : INT  := 75;	//CARRIAGE CONSTANT, DECELERATION
   SPARE_142 : INT ;
   OLD_CARR_POS_TO_ALARM : INT ;	//OLD CARRIAGE POSITION, HELP TO ALARM 20
   CNT_CARR_CONVERT : INT ;	//COUNTER VALUE FROM CARRIAGE, MOVED FROM DB61.DBD6 (DI TO I)
   OLD_CARR_POS : INT ;	//VALUE FROM LAST STOP
   CNT_CARRIAGE_POSITION : INT ;	//AT BOTTOM=0, INCREASE UPWARDS
   PALLET_HEIGHT : INT ;	//PALLET HEIGHT
   LOWERST_OK_CUT : INT  := 20;	//LOWERST CARRIAGE POSITION OK TO CUT
   CARR_POS_HS : INT ;	//CARRIAGE POSITION HIGH SPEED IN WRAP CYCLE
   STOP_AFTER_PC : INT ;	//CARRIAGE STOP AFTER PHOTOCELL, UPWARDS TO POS
   CARR_DOWN_BEFORE_CUTV : INT ;	//CARRIAGE DOWN BEFORE CUTTING, TO POS
   CARR_HS_TO_RS : INT  := 10;	//CHANGES HIGH SPEED TO RESET SPEED
   SPARE_164 : INT ;
   SPARE_166 : INT ;
   PALLET_MEASURING : INT ;	//OPTION, PALLET POSITION - LENGTH MEASURING
   PALLET_STOP_MEASURING : INT ;	//OPTION, PALLET POSITION - LENGTH MEASURING
   LENGTH_MEASURING : INT  := 45;	//VALUE TO ADJUST STOP PALLET
   SPARE_174 : INT ;
   SPARE_176 : INT ;
   SPARE_178 : INT ;
   DIV_BIT : WORD ;	//FROM OP3
   PREVCYCLETIME : INT ;
   MINCYCLETIME : INT  := 99;
   MAXCYCLETIME : INT ;
   SPEEDFILMMAN : INT ;
   CNT_FILMCONSUMPTION : INT ;	//COUNTER FILM CONSUMPTION, NUMBER OF WRAPS AT FIRST CYLINDER x 390mm
   SPARE_192 : INT ;
   PALLETSSINCE : INT ;
   NUMBER_OF_FILMCYCLES : DINT  := L#100;	//NUMBER OF FILMCYCLES (=CUTTING)
   FILMCONSUMPTION_DM : INT ;	//FILMCONSUMPTION IN DM
   VALUE_FILMMOTOR : INT ;
   TURNTABLE_VALUT_AT_END : INT ;
  END_STRUCT ;	
BEGIN
   PRG_CHOICE_OP3 := 4;
   OLD_PRG_POINTER := 1;
   PRG_POINTER := 1;
   FILMTENSION_TOP := 10;
   FILMTENSION_MIDDLE := 10;
   FILMTENSION_BOTTOM := 10;
   SET_POINT_TOPWRAP := 1;
   SET_POINT_BOTTOMWRAP := 2;
   SET_POINT_MS_TO_LS_TT := 66;
   SET_POINT_MID_SPEED_TT := 40;
   SET_POINT_HI_SPEED_TT := 55;
   SET_POINT_WRA_SPEED_DOWN := 35;
   SET_POINT_WRAPP_SPEED_UP := 35;
   SET_POINT_HI_SPEED_CARR := 100;
   CARR_STOP_AFTER_PC := 1;
   FILMWELDIND_TIME := S5T#180MS;
   SET_POINT_CONT_BEFORE_HS := 24;
   TT_SYNC_M_TO_L_90 := 42;
   RET_TURNTABLE := 95;
   TW_USED := 100;
   BW_USED := 200;
   FILMHOLDER_HOME := 125;
   OK_TO_SYNC_TURNTABLE := 20;
   VALUE_CLUTCH_OFF := 50;
   TT_LOW_SPEED := 6;
   TT_CONV_SPEED := 25;
   FFS_END_LEVEL := 2000;
   FFS_START_LEVEL := 4000;
   FFS_STEPS := 100;
   CONVEYOR_STOP_T0 := S5T#3S250MS;
   OUTFEEDING_TIME_T1 := S5T#500MS;
   DELAY_MOTOR_TO_CLUTCH_T2 := S5T#100MS;
   DELAY_FC_START_T3 := S5T#100MS;
   FILTER_S1254_PALLET_H_T4 := S5T#300MS;
   CLAMP_T5 := S5T#100MS;
   CUTTING_T6 := S5T#3S;
   KNIFEARM_BACK_T7 := S5T#2S;
   ALARMLONGCYCLE := S5T#1M30S;
   FILMHOLDER_CLOSE_T9 := S5T#1S;
   KNIFE_UP_T10 := S5T#400MS;
   CUTTING_ARM_HOME_T11 := S5T#1S;
   T12_DELAY_TT_STOP_0 := S5T#300MS;
   T51_T53_DELAY_TIME := S5T#250MS;
   T16_TIME_MS_TO_90 := S5T#1S500MS;
   ALARMLONGCONV1 := S5T#45S;
   RET_HISS := 75;
   CNT_CARRIAGE_POSITION := 8;
   PALLET_HEIGHT := 200;
   LOWERST_OK_CUT := 20;
   CARR_DOWN_BEFORE_CUTV := 6;
   CARR_HS_TO_RS := 10;
   PALLET_MEASURING := 413;
   LENGTH_MEASURING := 45;
   PREVCYCLETIME := 8;
   MINCYCLETIME := 5;
   MAXCYCLETIME := 29;
   NUMBER_OF_FILMCYCLES := L#100;
   VALUE_FILMMOTOR := 4000;
END_DATA_BLOCK

DATA_BLOCK "EDITING_PROG"	// DB 13
AUTHOR : LKA
NAME : MAINDATA
VERSION : 0.1
  STRUCT
   PRG_CHOICE_OP3 : INT  := 1;	//PROGRAMME CHOICE FROM OP3
   EXTERNAL_PROGRAMME : INT ;	//EXTERNAL PROGRAMME CHOICE
   OLD_PRG_POINTER : INT ;	//OLD PROGRAMME VALUE
   PRG_POINTER : INT  := 1;	//PROGRAMME WHICH PARAMETR IS TO BE CHANGED
   ACTUAL_PROGRAMME : INT ;	//AKTUELLT PROGRAM SOM ANVÄNDS I FILMCYKELN
   ACTUAL_PROGRAMME_JUMP : INT ;	//JUMP VALUE TO FC 21-29
   SPARE_12 : INT ;
   SPARE_14 : INT ;
   FILMTENSION_TOP : INT  := 10;	//SET POINT FILMTENSION TOP
   FILMTENSION_MIDDLE : INT  := 10;	//SET POINT FILMTENSION MIDDLE
   FILMTENSION_BOTTOM : INT  := 10;	//SET POINT FILMTENSION BOTTOM
   SET_POINT_TOPWRAP : INT  := 1;	//SET POINT NUMBER OF TOPWRAP
   SET_POINT_BOTTOMWRAP : INT  := 2;	//SET POINT NUMBER OF BOTTOMWRAP
   SET_POINT_MS_TO_LS_TT : INT  := 66;
   SET_POINT_MID_SPEED_TT : INT  := 40;	//SET POINT MEDDLE SPEED, TURNTABLE
   SET_POINT_HI_SPEED_TT : INT  := 55;	//SET POINT HIGH SPEED, TURNTABLE
   SET_POINT_WRA_SPEED_DOWN : INT  := 35;	//SET POINT WRAPPING SPEED DOWNWARDS, CARRIAGE
   SET_POINT_WRAPP_SPEED_UP : INT  := 35;	//SET POINT WRAPPING SPEED UPWARDS, CARRIAGE
   SET_POINT_HI_SPEED_CARR : INT  := 100;	//SET POINT HIGH SPEED, CARRIAGE
   TOP_PLATE : BOOL  := TRUE;	//PROGRAMME LAY OUT TOP PLATE
   TOP_FILM : BOOL ;	//PROGRAMME LAY OUT TOP FILM
   WATERPROFE_TOP_FILM : BOOL ;	//PROGRAMME LAY OUT LOADCASSETTE
   FILMWELDING : BOOL  := TRUE;	//PROGRAMME LAY OUT FILMWELDING
   HOT_AIR_FILMWELDING : BOOL ;	//PROGRAMME LAY OUT HOT AIR FILMWELDING
   SPARE_40 : INT ;
   SPARE_42 : INT ;
   SPARE_44 : INT ;
   CARR_STOP_AFTER_PC : INT ;	//CARRIAGE STOP AFTER PHOTOCELL
   CARR_DOWN_BEFORE_CUT : INT ;	//CARRIAGE DOWN BEFORE CUTTING
   FILMWELDIND_TIME : S5TIME  := S5T#400MS;	//FILMWELDING TIME
   SET_POINT_CONT_BEFORE_HS : INT  := 100;	//SET POINT PULSES BEFORE HIGH SPEED
   SPARE_54 : INT ;
   SPARE_56 : INT ;
   SPARE_58 : INT ;
   CONVEYORING_IN : BOOL  := TRUE;	//PROGRAMME CONFIGURATION, CONVEYING IN, LEFT=0, RIGHT=1
   IN_90 : BOOL ;	//PROGRAMME CONFIGURATION, 90 DEGREE INFEEDING
   OUT_90 : BOOL ;	//PROGRAMME CONFIGURATION, 90 DEGREE OUTFEEDING
   HALF_PALLET : BOOL ;	//PROGRAMME CONFIGURATION, HALF PALLET INDICATING
   PALLET_LENGTH : BOOL ;	//PROGRAMME CONFIGURATION, PALLET LENGTH MEASURING
   ENABLE_TOPPLATE : BOOL  := TRUE;	//PROGRAMME CONFIGURATION, RUN TOPPLATE FC
   NO_FILM : BOOL ;	//PROGRAMME CONFIGURATION, TEST FUNCTION PROGRAMME WITHOUT FILM
   NO_CONVEYORING : BOOL ;	//PROGRAMME CONFIGURATION, TEST FUNCTION PROGRAMME WITHOUT CONVEYORING
   SOFT_RAMP_CONV : BOOL ;	//PROGRAMME CONFIGURATION, SOFT RAMP IN CONVEYORING SPEED
   FFS_OFF : BOOL ;	//PROG CONFIG, 1= EASY FILM FEED SYSTEM, NO SELF FINDING BY MACHINE
   TYPE_OFF_WELDING : BOOL ;	//PROGRAMME CONFIGURATION, 0= BT WELDING, 1= HOT AIR WELDING
   HALF_IN_OUT_FEED_S : BOOL  := TRUE;	//PROG CONFIG, HALF IN AND OUT CONVEYING SIMULTANEOUS
   IN_OUT_FEED_SIMULTAN : BOOL ;	//PROG CONFIG, IN AND OUT CONVEYING SIMULTANEOUS
   SIGNAL_EXTERNAL : BOOL ;	//CONVEYING PAUSED THEN NO SIGNAL, S11 OR S13
   SPARE_62 : INT ;
  END_STRUCT ;	
BEGIN
   PRG_CHOICE_OP3 := 1;
   PRG_POINTER := 1;
   FILMTENSION_TOP := 10;
   FILMTENSION_MIDDLE := 10;
   FILMTENSION_BOTTOM := 10;
   SET_POINT_TOPWRAP := 1;
   SET_POINT_BOTTOMWRAP := 2;
   SET_POINT_MS_TO_LS_TT := 66;
   SET_POINT_MID_SPEED_TT := 40;
   SET_POINT_HI_SPEED_TT := 55;
   SET_POINT_WRA_SPEED_DOWN := 35;
   SET_POINT_WRAPP_SPEED_UP := 35;
   SET_POINT_HI_SPEED_CARR := 100;
   TOP_PLATE := TRUE;
   FILMWELDING := TRUE;
   FILMWELDIND_TIME := S5T#400MS;
   SET_POINT_CONT_BEFORE_HS := 100;
   CONVEYORING_IN := TRUE;
   ENABLE_TOPPLATE := TRUE;
   HALF_IN_OUT_FEED_S := TRUE;
END_DATA_BLOCK

DATA_BLOCK "PROG_1_DATA"	// DB 21
AUTHOR : LKA
NAME : MAINDATA
VERSION : 0.1
  STRUCT
   PRG_CHOICE_OP3 : INT  := 1;	//PROGRAMME CHOICE FROM OP3
   EXTERNAL_PROGRAMME : INT ;	//EXTERNAL PROGRAMME CHOICE
   OLD_PRG_POINTER : INT ;	//OLD PROGRAMME VALUE
   PRG_POINTER : INT  := 1;	//PROGRAMME WHICH PARAMETR IS TO BE CHANGED
   ACTUAL_PROGRAMME : INT ;	//AKTUELLT PROGRAM SOM ANVÄNDS I FILMCYKELN
   ACTUAL_PROGRAMME_JUMP : INT ;	//JUMP VALUE TO FC 21-29
   SPARE_12 : INT ;
   SPARE_14 : INT ;
   FILMTENSION_TOP : INT  := 10;	//SET POINT FILMTENSION TOP
   FILMTENSION_MIDDLE : INT  := 10;	//SET POINT FILMTENSION MIDDLE
   FILMTENSION_BOTTOM : INT  := 10;	//SET POINT FILMTENSION BOTTOM
   SET_POINT_TOPWRAP : INT  := 1;	//SET POINT NUMBER OF TOPWRAP
   SET_POINT_BOTTOMWRAP : INT  := 2;	//SET POINT NUMBER OF BOTTOMWRAP
   SET_POINT_MS_TO_LS_TT : INT  := 66;
   SET_POINT_MID_SPEED_TT : INT  := 40;	//SET POINT MEDDLE SPEED, TURNTABLE
   SET_POINT_HI_SPEED_TT : INT  := 55;	//SET POINT HIGH SPEED, TURNTABLE
   SET_POINT_WRA_SPEED_DOWN : INT  := 35;	//SET POINT WRAPPING SPEED DOWNWARDS, CARRIAGE
   SET_POINT_WRAPP_SPEED_UP : INT  := 35;	//SET POINT WRAPPING SPEED UPWARDS, CARRIAGE
   SET_POINT_HI_SPEED_CARR : INT  := 100;	//SET POINT HIGH SPEED, CARRIAGE
   TOP_PLATE : BOOL ;	//PROGRAMME LAY OUT TOP PLATE
   TOP_FILM : BOOL ;	//PROGRAMME LAY OUT TOP FILM
   WATERPROFE_TOP_FILM : BOOL ;	//PROGRAMME LAY OUT LOADCASSETTE
   FILMWELDING : BOOL ;	//PROGRAMME LAY OUT FILMWELDING
   HOT_AIR_FILMWELDING : BOOL ;	//PROGRAMME LAY OUT HOT AIR FILMWELDING
   SPARE_40 : INT ;
   SPARE_42 : INT ;
   SPARE_44 : INT ;
   CARR_STOP_AFTER_PC : INT  := 1;	//CARRIAGE STOP AFTER PHOTOCELL
   CARR_DOWN_BEFORE_CUT : INT ;	//CARRIAGE DOWN BEFORE CUTTING
   FILMWELDIND_TIME : S5TIME  := S5T#400MS;	//FILMWELDING TIME
   SET_POINT_CONT_BEFORE_HS : INT  := 100;	//SET POINT PULSES BEFORE HIGH SPEED
   SPARE_54 : INT ;
   SPARE_56 : INT ;
  END_STRUCT ;	
BEGIN
   PRG_CHOICE_OP3 := 1;
   PRG_POINTER := 1;
   FILMTENSION_TOP := 10;
   FILMTENSION_MIDDLE := 10;
   FILMTENSION_BOTTOM := 10;
   SET_POINT_TOPWRAP := 1;
   SET_POINT_BOTTOMWRAP := 2;
   SET_POINT_MS_TO_LS_TT := 66;
   SET_POINT_MID_SPEED_TT := 40;
   SET_POINT_HI_SPEED_TT := 55;
   SET_POINT_WRA_SPEED_DOWN := 35;
   SET_POINT_WRAPP_SPEED_UP := 35;
   SET_POINT_HI_SPEED_CARR := 100;
   CARR_STOP_AFTER_PC := 1;
   FILMWELDIND_TIME := S5T#400MS;
   SET_POINT_CONT_BEFORE_HS := 100;
END_DATA_BLOCK

DATA_BLOCK "PROG_2_DATA"	// DB 22
AUTHOR : LKA
NAME : MAINDATA
VERSION : 0.1
  STRUCT
   PRG_CHOICE_OP3 : INT  := 1;	//PROGRAMME CHOICE FROM OP3
   EXTERNAL_PROGRAMME : INT ;	//EXTERNAL PROGRAMME CHOICE
   OLD_PRG_POINTER : INT ;	//OLD PROGRAMME VALUE
   PRG_POINTER : INT  := 1;	//PROGRAMME WHICH PARAMETR IS TO BE CHANGED
   ACTUAL_PROGRAMME : INT ;	//AKTUELLT PROGRAM SOM ANVÄNDS I FILMCYKELN
   ACTUAL_PROGRAMME_JUMP : INT ;	//JUMP VALUE TO FC 21-29
   SPARE_12 : INT ;
   SPARE_14 : INT ;
   FILMTENSION_TOP : INT  := 10;	//SET POINT FILMTENSION TOP
   FILMTENSION_MIDDLE : INT  := 10;	//SET POINT FILMTENSION MIDDLE
   FILMTENSION_BOTTOM : INT  := 10;	//SET POINT FILMTENSION BOTTOM
   SET_POINT_TOPWRAP : INT  := 1;	//SET POINT NUMBER OF TOPWRAP
   SET_POINT_BOTTOMWRAP : INT  := 2;	//SET POINT NUMBER OF BOTTOMWRAP
   SET_POINT_MS_TO_LS_TT : INT  := 66;
   SET_POINT_MID_SPEED_TT : INT  := 40;	//SET POINT MEDDLE SPEED, TURNTABLE
   SET_POINT_HI_SPEED_TT : INT  := 55;	//SET POINT HIGH SPEED, TURNTABLE
   SET_POINT_WRA_SPEED_DOWN : INT  := 35;	//SET POINT WRAPPING SPEED DOWNWARDS, CARRIAGE
   SET_POINT_WRAPP_SPEED_UP : INT  := 35;	//SET POINT WRAPPING SPEED UPWARDS, CARRIAGE
   SET_POINT_HI_SPEED_CARR : INT  := 100;	//SET POINT HIGH SPEED, CARRIAGE
   TOP_PLATE : BOOL ;	//PROGRAMME LAY OUT TOP PLATE
   TOP_FILM : BOOL ;	//PROGRAMME LAY OUT TOP FILM
   WATERPROFE_TOP_FILM : BOOL ;	//PROGRAMME LAY OUT LOADCASSETTE
   FILMWELDING : BOOL ;	//PROGRAMME LAY OUT FILMWELDING
   HOT_AIR_FILMWELDING : BOOL ;	//PROGRAMME LAY OUT HOT AIR FILMWELDING
   SPARE_40 : INT ;
   SPARE_42 : INT ;
   SPARE_44 : INT ;
   CARR_STOP_AFTER_PC : INT  := 1;	//CARRIAGE STOP AFTER PHOTOCELL
   CARR_DOWN_BEFORE_CUT : INT ;	//CARRIAGE DOWN BEFORE CUTTING
   FILMWELDIND_TIME : S5TIME  := S5T#400MS;	//FILMWELDING TIME
   SET_POINT_CONT_BEFORE_HS : INT  := 100;	//SET POINT PULSES BEFORE HIGH SPEED
   SPARE_54 : INT ;
   SPARE_56 : INT ;
  END_STRUCT ;	
BEGIN
   PRG_CHOICE_OP3 := 1;
   PRG_POINTER := 1;
   FILMTENSION_TOP := 10;
   FILMTENSION_MIDDLE := 10;
   FILMTENSION_BOTTOM := 10;
   SET_POINT_TOPWRAP := 1;
   SET_POINT_BOTTOMWRAP := 2;
   SET_POINT_MS_TO_LS_TT := 66;
   SET_POINT_MID_SPEED_TT := 40;
   SET_POINT_HI_SPEED_TT := 55;
   SET_POINT_WRA_SPEED_DOWN := 35;
   SET_POINT_WRAPP_SPEED_UP := 35;
   SET_POINT_HI_SPEED_CARR := 100;
   FILMWELDING := TRUE;
   CARR_STOP_AFTER_PC := 1;
   FILMWELDIND_TIME := S5T#400MS;
   SET_POINT_CONT_BEFORE_HS := 100;
END_DATA_BLOCK

DATA_BLOCK "PROG_3_DATA"	// DB 23
AUTHOR : LKA
NAME : MAINDATA
VERSION : 0.1
  STRUCT
   PRG_CHOICE_OP3 : INT  := 1;	//PROGRAMME CHOICE FROM OP3
   EXTERNAL_PROGRAMME : INT ;	//EXTERNAL PROGRAMME CHOICE
   OLD_PRG_POINTER : INT ;	//OLD PROGRAMME VALUE
   PRG_POINTER : INT  := 1;	//PROGRAMME WHICH PARAMETR IS TO BE CHANGED
   ACTUAL_PROGRAMME : INT ;	//AKTUELLT PROGRAM SOM ANVÄNDS I FILMCYKELN
   ACTUAL_PROGRAMME_JUMP : INT ;	//JUMP VALUE TO FC 21-29
   SPARE_12 : INT ;
   SPARE_14 : INT ;
   FILMTENSION_TOP : INT  := 10;	//SET POINT FILMTENSION TOP
   FILMTENSION_MIDDLE : INT  := 10;	//SET POINT FILMTENSION MIDDLE
   FILMTENSION_BOTTOM : INT  := 10;	//SET POINT FILMTENSION BOTTOM
   SET_POINT_TOPWRAP : INT  := 2;	//SET POINT NUMBER OF TOPWRAP
   SET_POINT_BOTTOMWRAP : INT  := 3;	//SET POINT NUMBER OF BOTTOMWRAP
   SET_POINT_MS_TO_LS_TT : INT  := 66;
   SET_POINT_MID_SPEED_TT : INT  := 40;	//SET POINT MEDDLE SPEED, TURNTABLE
   SET_POINT_HI_SPEED_TT : INT  := 55;	//SET POINT HIGH SPEED, TURNTABLE
   SET_POINT_WRA_SPEED_DOWN : INT  := 35;	//SET POINT WRAPPING SPEED DOWNWARDS, CARRIAGE
   SET_POINT_WRAPP_SPEED_UP : INT  := 35;	//SET POINT WRAPPING SPEED UPWARDS, CARRIAGE
   SET_POINT_HI_SPEED_CARR : INT  := 100;	//SET POINT HIGH SPEED, CARRIAGE
   TOP_PLATE : BOOL ;	//PROGRAMME LAY OUT TOP PLATE
   TOP_FILM : BOOL ;	//PROGRAMME LAY OUT TOP FILM
   WATERPROFE_TOP_FILM : BOOL ;	//PROGRAMME LAY OUT LOADCASSETTE
   FILMWELDING : BOOL ;	//PROGRAMME LAY OUT FILMWELDING
   HOT_AIR_FILMWELDING : BOOL ;	//PROGRAMME LAY OUT HOT AIR FILMWELDING
   SPARE_40 : INT ;
   SPARE_42 : INT ;
   SPARE_44 : INT ;
   CARR_STOP_AFTER_PC : INT  := 5;	//CARRIAGE STOP AFTER PHOTOCELL
   CARR_DOWN_BEFORE_CUT : INT  := 999;	//CARRIAGE DOWN BEFORE CUTTING
   FILMWELDIND_TIME : S5TIME  := S5T#400MS;	//FILMWELDING TIME
   SET_POINT_CONT_BEFORE_HS : INT  := 100;	//SET POINT PULSES BEFORE HIGH SPEED
   SPARE_54 : INT ;
   SPARE_56 : INT ;
  END_STRUCT ;	
BEGIN
   PRG_CHOICE_OP3 := 1;
   PRG_POINTER := 1;
   FILMTENSION_TOP := 10;
   FILMTENSION_MIDDLE := 10;
   FILMTENSION_BOTTOM := 10;
   SET_POINT_TOPWRAP := 2;
   SET_POINT_BOTTOMWRAP := 3;
   SET_POINT_MS_TO_LS_TT := 66;
   SET_POINT_MID_SPEED_TT := 40;
   SET_POINT_HI_SPEED_TT := 55;
   SET_POINT_WRA_SPEED_DOWN := 35;
   SET_POINT_WRAPP_SPEED_UP := 35;
   SET_POINT_HI_SPEED_CARR := 100;
   FILMWELDING := TRUE;
   CARR_STOP_AFTER_PC := 5;
   CARR_DOWN_BEFORE_CUT := 999;
   FILMWELDIND_TIME := S5T#400MS;
   SET_POINT_CONT_BEFORE_HS := 100;
END_DATA_BLOCK

DATA_BLOCK "PROG_4_DATA"	// DB 24
AUTHOR : LKA
NAME : MAINDATA
VERSION : 0.1
  STRUCT
   PRG_CHOICE_OP3 : INT  := 1;	//PROGRAMME CHOICE FROM OP3
   EXTERNAL_PROGRAMME : INT ;	//EXTERNAL PROGRAMME CHOICE
   OLD_PRG_POINTER : INT ;	//OLD PROGRAMME VALUE
   PRG_POINTER : INT  := 1;	//PROGRAMME WHICH PARAMETR IS TO BE CHANGED
   ACTUAL_PROGRAMME : INT ;	//AKTUELLT PROGRAM SOM ANVÄNDS I FILMCYKELN
   ACTUAL_PROGRAMME_JUMP : INT ;	//JUMP VALUE TO FC 21-29
   SPARE_12 : INT ;
   SPARE_14 : INT ;
   FILMTENSION_TOP : INT  := 10;	//SET POINT FILMTENSION TOP
   FILMTENSION_MIDDLE : INT  := 10;	//SET POINT FILMTENSION MIDDLE
   FILMTENSION_BOTTOM : INT  := 10;	//SET POINT FILMTENSION BOTTOM
   SET_POINT_TOPWRAP : INT  := 1;	//SET POINT NUMBER OF TOPWRAP
   SET_POINT_BOTTOMWRAP : INT  := 2;	//SET POINT NUMBER OF BOTTOMWRAP
   SET_POINT_MS_TO_LS_TT : INT  := 66;
   SET_POINT_MID_SPEED_TT : INT  := 40;	//SET POINT MEDDLE SPEED, TURNTABLE
   SET_POINT_HI_SPEED_TT : INT  := 55;	//SET POINT HIGH SPEED, TURNTABLE
   SET_POINT_WRA_SPEED_DOWN : INT  := 35;	//SET POINT WRAPPING SPEED DOWNWARDS, CARRIAGE
   SET_POINT_WRAPP_SPEED_UP : INT  := 35;	//SET POINT WRAPPING SPEED UPWARDS, CARRIAGE
   SET_POINT_HI_SPEED_CARR : INT  := 100;	//SET POINT HIGH SPEED, CARRIAGE
   TOP_PLATE : BOOL ;	//PROGRAMME LAY OUT TOP PLATE
   TOP_FILM : BOOL ;	//PROGRAMME LAY OUT TOP FILM
   WATERPROFE_TOP_FILM : BOOL ;	//PROGRAMME LAY OUT LOADCASSETTE
   FILMWELDING : BOOL ;	//PROGRAMME LAY OUT FILMWELDING
   HOT_AIR_FILMWELDING : BOOL ;	//PROGRAMME LAY OUT HOT AIR FILMWELDING
   SPARE_40 : INT ;
   SPARE_42 : INT ;
   SPARE_44 : INT ;
   CARR_STOP_AFTER_PC : INT  := 1;	//CARRIAGE STOP AFTER PHOTOCELL
   CARR_DOWN_BEFORE_CUT : INT ;	//CARRIAGE DOWN BEFORE CUTTING
   FILMWELDIND_TIME : S5TIME  := S5T#180MS;	//FILMWELDING TIME
   SET_POINT_CONT_BEFORE_HS : INT  := 24;	//SET POINT PULSES BEFORE HIGH SPEED
   SPARE_54 : INT ;
   SPARE_56 : INT ;
  END_STRUCT ;	
BEGIN
   PRG_CHOICE_OP3 := 1;
   PRG_POINTER := 1;
   FILMTENSION_TOP := 10;
   FILMTENSION_MIDDLE := 10;
   FILMTENSION_BOTTOM := 10;
   SET_POINT_TOPWRAP := 1;
   SET_POINT_BOTTOMWRAP := 2;
   SET_POINT_MS_TO_LS_TT := 66;
   SET_POINT_MID_SPEED_TT := 40;
   SET_POINT_HI_SPEED_TT := 55;
   SET_POINT_WRA_SPEED_DOWN := 35;
   SET_POINT_WRAPP_SPEED_UP := 35;
   SET_POINT_HI_SPEED_CARR := 100;
   CARR_STOP_AFTER_PC := 1;
   FILMWELDIND_TIME := S5T#180MS;
   SET_POINT_CONT_BEFORE_HS := 24;
END_DATA_BLOCK

DATA_BLOCK "PROG_5_DATA"	// DB 25
AUTHOR : LKA
NAME : MAINDATA
VERSION : 0.1
  STRUCT
   PRG_CHOICE_OP3 : INT  := 1;	//PROGRAMME CHOICE FROM OP3
   EXTERNAL_PROGRAMME : INT ;	//EXTERNAL PROGRAMME CHOICE
   OLD_PRG_POINTER : INT ;	//OLD PROGRAMME VALUE
   PRG_POINTER : INT  := 1;	//PROGRAMME WHICH PARAMETR IS TO BE CHANGED
   ACTUAL_PROGRAMME : INT ;	//AKTUELLT PROGRAM SOM ANVÄNDS I FILMCYKELN
   ACTUAL_PROGRAMME_JUMP : INT ;	//JUMP VALUE TO FC 21-29
   SPARE_12 : INT ;
   SPARE_14 : INT ;
   FILMTENSION_TOP : INT  := 10;	//SET POINT FILMTENSION TOP
   FILMTENSION_MIDDLE : INT  := 10;	//SET POINT FILMTENSION MIDDLE
   FILMTENSION_BOTTOM : INT  := 10;	//SET POINT FILMTENSION BOTTOM
   SET_POINT_TOPWRAP : INT  := 1;	//SET POINT NUMBER OF TOPWRAP
   SET_POINT_BOTTOMWRAP : INT  := 2;	//SET POINT NUMBER OF BOTTOMWRAP
   SET_POINT_MS_TO_LS_TT : INT  := 66;
   SET_POINT_MID_SPEED_TT : INT  := 40;	//SET POINT MEDDLE SPEED, TURNTABLE
   SET_POINT_HI_SPEED_TT : INT  := 55;	//SET POINT HIGH SPEED, TURNTABLE
   SET_POINT_WRA_SPEED_DOWN : INT  := 35;	//SET POINT WRAPPING SPEED DOWNWARDS, CARRIAGE
   SET_POINT_WRAPP_SPEED_UP : INT  := 35;	//SET POINT WRAPPING SPEED UPWARDS, CARRIAGE
   SET_POINT_HI_SPEED_CARR : INT  := 100;	//SET POINT HIGH SPEED, CARRIAGE
   TOP_PLATE : BOOL ;	//PROGRAMME LAY OUT TOP PLATE
   TOP_FILM : BOOL ;	//PROGRAMME LAY OUT TOP FILM
   WATERPROFE_TOP_FILM : BOOL ;	//PROGRAMME LAY OUT LOADCASSETTE
   FILMWELDING : BOOL ;	//PROGRAMME LAY OUT FILMWELDING
   HOT_AIR_FILMWELDING : BOOL ;	//PROGRAMME LAY OUT HOT AIR FILMWELDING
   SPARE_40 : INT ;
   SPARE_42 : INT ;
   SPARE_44 : INT ;
   CARR_STOP_AFTER_PC : INT  := 1;	//CARRIAGE STOP AFTER PHOTOCELL
   CARR_DOWN_BEFORE_CUT : INT ;	//CARRIAGE DOWN BEFORE CUTTING
   FILMWELDIND_TIME : S5TIME  := S5T#180MS;	//FILMWELDING TIME
   SET_POINT_CONT_BEFORE_HS : INT  := 24;	//SET POINT PULSES BEFORE HIGH SPEED
   SPARE_54 : INT ;
   SPARE_56 : INT ;
  END_STRUCT ;	
BEGIN
   PRG_CHOICE_OP3 := 1;
   PRG_POINTER := 1;
   FILMTENSION_TOP := 10;
   FILMTENSION_MIDDLE := 10;
   FILMTENSION_BOTTOM := 10;
   SET_POINT_TOPWRAP := 1;
   SET_POINT_BOTTOMWRAP := 2;
   SET_POINT_MS_TO_LS_TT := 66;
   SET_POINT_MID_SPEED_TT := 40;
   SET_POINT_HI_SPEED_TT := 55;
   SET_POINT_WRA_SPEED_DOWN := 35;
   SET_POINT_WRAPP_SPEED_UP := 35;
   SET_POINT_HI_SPEED_CARR := 100;
   CARR_STOP_AFTER_PC := 1;
   FILMWELDIND_TIME := S5T#180MS;
   SET_POINT_CONT_BEFORE_HS := 24;
END_DATA_BLOCK

DATA_BLOCK "PROG_6_DATA"	// DB 26
AUTHOR : LKA
NAME : MAINDATA
VERSION : 0.1
  STRUCT
   PRG_CHOICE_OP3 : INT  := 1;	//PROGRAMME CHOICE FROM OP3
   EXTERNAL_PROGRAMME : INT ;	//EXTERNAL PROGRAMME CHOICE
   OLD_PRG_POINTER : INT ;	//OLD PROGRAMME VALUE
   PRG_POINTER : INT  := 1;	//PROGRAMME WHICH PARAMETR IS TO BE CHANGED
   ACTUAL_PROGRAMME : INT ;	//AKTUELLT PROGRAM SOM ANVÄNDS I FILMCYKELN
   ACTUAL_PROGRAMME_JUMP : INT ;	//JUMP VALUE TO FC 21-29
   SPARE_12 : INT ;
   SPARE_14 : INT ;
   FILMTENSION_TOP : INT  := 10;	//SET POINT FILMTENSION TOP
   FILMTENSION_MIDDLE : INT  := 10;	//SET POINT FILMTENSION MIDDLE
   FILMTENSION_BOTTOM : INT  := 10;	//SET POINT FILMTENSION BOTTOM
   SET_POINT_TOPWRAP : INT  := 1;	//SET POINT NUMBER OF TOPWRAP
   SET_POINT_BOTTOMWRAP : INT  := 2;	//SET POINT NUMBER OF BOTTOMWRAP
   SET_POINT_MS_TO_LS_TT : INT  := 66;
   SET_POINT_MID_SPEED_TT : INT  := 40;	//SET POINT MEDDLE SPEED, TURNTABLE
   SET_POINT_HI_SPEED_TT : INT  := 55;	//SET POINT HIGH SPEED, TURNTABLE
   SET_POINT_WRA_SPEED_DOWN : INT  := 35;	//SET POINT WRAPPING SPEED DOWNWARDS, CARRIAGE
   SET_POINT_WRAPP_SPEED_UP : INT  := 35;	//SET POINT WRAPPING SPEED UPWARDS, CARRIAGE
   SET_POINT_HI_SPEED_CARR : INT  := 100;	//SET POINT HIGH SPEED, CARRIAGE
   TOP_PLATE : BOOL ;	//PROGRAMME LAY OUT TOP PLATE
   TOP_FILM : BOOL ;	//PROGRAMME LAY OUT TOP FILM
   WATERPROFE_TOP_FILM : BOOL ;	//PROGRAMME LAY OUT LOADCASSETTE
   FILMWELDING : BOOL ;	//PROGRAMME LAY OUT FILMWELDING
   HOT_AIR_FILMWELDING : BOOL ;	//PROGRAMME LAY OUT HOT AIR FILMWELDING
   SPARE_40 : INT ;
   SPARE_42 : INT ;
   SPARE_44 : INT ;
   CARR_STOP_AFTER_PC : INT  := 1;	//CARRIAGE STOP AFTER PHOTOCELL
   CARR_DOWN_BEFORE_CUT : INT ;	//CARRIAGE DOWN BEFORE CUTTING
   FILMWELDIND_TIME : S5TIME  := S5T#180MS;	//FILMWELDING TIME
   SET_POINT_CONT_BEFORE_HS : INT  := 24;	//SET POINT PULSES BEFORE HIGH SPEED
   SPARE_54 : INT ;
   SPARE_56 : INT ;
  END_STRUCT ;	
BEGIN
   PRG_CHOICE_OP3 := 1;
   PRG_POINTER := 1;
   FILMTENSION_TOP := 10;
   FILMTENSION_MIDDLE := 10;
   FILMTENSION_BOTTOM := 10;
   SET_POINT_TOPWRAP := 1;
   SET_POINT_BOTTOMWRAP := 2;
   SET_POINT_MS_TO_LS_TT := 66;
   SET_POINT_MID_SPEED_TT := 40;
   SET_POINT_HI_SPEED_TT := 55;
   SET_POINT_WRA_SPEED_DOWN := 35;
   SET_POINT_WRAPP_SPEED_UP := 35;
   SET_POINT_HI_SPEED_CARR := 100;
   CARR_STOP_AFTER_PC := 1;
   FILMWELDIND_TIME := S5T#180MS;
   SET_POINT_CONT_BEFORE_HS := 24;
END_DATA_BLOCK

DATA_BLOCK "PROG_7_DATA"	// DB 27
AUTHOR : LKA
NAME : MAINDATA
VERSION : 0.1
  STRUCT
   PRG_CHOICE_OP3 : INT  := 1;	//PROGRAMME CHOICE FROM OP3
   EXTERNAL_PROGRAMME : INT ;	//EXTERNAL PROGRAMME CHOICE
   OLD_PRG_POINTER : INT ;	//OLD PROGRAMME VALUE
   PRG_POINTER : INT  := 1;	//PROGRAMME WHICH PARAMETR IS TO BE CHANGED
   ACTUAL_PROGRAMME : INT ;	//AKTUELLT PROGRAM SOM ANVÄNDS I FILMCYKELN
   ACTUAL_PROGRAMME_JUMP : INT ;	//JUMP VALUE TO FC 21-29
   SPARE_12 : INT ;
   SPARE_14 : INT ;
   FILMTENSION_TOP : INT  := 10;	//SET POINT FILMTENSION TOP
   FILMTENSION_MIDDLE : INT  := 10;	//SET POINT FILMTENSION MIDDLE
   FILMTENSION_BOTTOM : INT  := 10;	//SET POINT FILMTENSION BOTTOM
   SET_POINT_TOPWRAP : INT  := 1;	//SET POINT NUMBER OF TOPWRAP
   SET_POINT_BOTTOMWRAP : INT  := 2;	//SET POINT NUMBER OF BOTTOMWRAP
   SET_POINT_MS_TO_LS_TT : INT  := 66;
   SET_POINT_MID_SPEED_TT : INT  := 40;	//SET POINT MEDDLE SPEED, TURNTABLE
   SET_POINT_HI_SPEED_TT : INT  := 55;	//SET POINT HIGH SPEED, TURNTABLE
   SET_POINT_WRA_SPEED_DOWN : INT  := 35;	//SET POINT WRAPPING SPEED DOWNWARDS, CARRIAGE
   SET_POINT_WRAPP_SPEED_UP : INT  := 35;	//SET POINT WRAPPING SPEED UPWARDS, CARRIAGE
   SET_POINT_HI_SPEED_CARR : INT  := 100;	//SET POINT HIGH SPEED, CARRIAGE
   TOP_PLATE : BOOL ;	//PROGRAMME LAY OUT TOP PLATE
   TOP_FILM : BOOL ;	//PROGRAMME LAY OUT TOP FILM
   WATERPROFE_TOP_FILM : BOOL ;	//PROGRAMME LAY OUT LOADCASSETTE
   FILMWELDING : BOOL ;	//PROGRAMME LAY OUT FILMWELDING
   HOT_AIR_FILMWELDING : BOOL ;	//PROGRAMME LAY OUT HOT AIR FILMWELDING
   SPARE_40 : INT ;
   SPARE_42 : INT ;
   SPARE_44 : INT ;
   CARR_STOP_AFTER_PC : INT  := 1;	//CARRIAGE STOP AFTER PHOTOCELL
   CARR_DOWN_BEFORE_CUT : INT ;	//CARRIAGE DOWN BEFORE CUTTING
   FILMWELDIND_TIME : S5TIME  := S5T#180MS;	//FILMWELDING TIME
   SET_POINT_CONT_BEFORE_HS : INT  := 24;	//SET POINT PULSES BEFORE HIGH SPEED
   SPARE_54 : INT ;
   SPARE_56 : INT ;
  END_STRUCT ;	
BEGIN
   PRG_CHOICE_OP3 := 1;
   PRG_POINTER := 1;
   FILMTENSION_TOP := 10;
   FILMTENSION_MIDDLE := 10;
   FILMTENSION_BOTTOM := 10;
   SET_POINT_TOPWRAP := 1;
   SET_POINT_BOTTOMWRAP := 2;
   SET_POINT_MS_TO_LS_TT := 66;
   SET_POINT_MID_SPEED_TT := 40;
   SET_POINT_HI_SPEED_TT := 55;
   SET_POINT_WRA_SPEED_DOWN := 35;
   SET_POINT_WRAPP_SPEED_UP := 35;
   SET_POINT_HI_SPEED_CARR := 100;
   CARR_STOP_AFTER_PC := 1;
   FILMWELDIND_TIME := S5T#180MS;
   SET_POINT_CONT_BEFORE_HS := 24;
END_DATA_BLOCK

DATA_BLOCK "PROG_8_DATA"	// DB 28
AUTHOR : LKA
NAME : MAINDATA
VERSION : 0.1
  STRUCT
   PRG_CHOICE_OP3 : INT  := 1;	//PROGRAMME CHOICE FROM OP3
   EXTERNAL_PROGRAMME : INT ;	//EXTERNAL PROGRAMME CHOICE
   OLD_PRG_POINTER : INT ;	//OLD PROGRAMME VALUE
   PRG_POINTER : INT  := 1;	//PROGRAMME WHICH PARAMETR IS TO BE CHANGED
   ACTUAL_PROGRAMME : INT ;	//AKTUELLT PROGRAM SOM ANVÄNDS I FILMCYKELN
   ACTUAL_PROGRAMME_JUMP : INT ;	//JUMP VALUE TO FC 21-29
   SPARE_12 : INT ;
   SPARE_14 : INT ;
   FILMTENSION_TOP : INT  := 10;	//SET POINT FILMTENSION TOP
   FILMTENSION_MIDDLE : INT  := 10;	//SET POINT FILMTENSION MIDDLE
   FILMTENSION_BOTTOM : INT  := 10;	//SET POINT FILMTENSION BOTTOM
   SET_POINT_TOPWRAP : INT  := 1;	//SET POINT NUMBER OF TOPWRAP
   SET_POINT_BOTTOMWRAP : INT  := 2;	//SET POINT NUMBER OF BOTTOMWRAP
   SET_POINT_MS_TO_LS_TT : INT  := 66;
   SET_POINT_MID_SPEED_TT : INT  := 40;	//SET POINT MEDDLE SPEED, TURNTABLE
   SET_POINT_HI_SPEED_TT : INT  := 55;	//SET POINT HIGH SPEED, TURNTABLE
   SET_POINT_WRA_SPEED_DOWN : INT  := 35;	//SET POINT WRAPPING SPEED DOWNWARDS, CARRIAGE
   SET_POINT_WRAPP_SPEED_UP : INT  := 35;	//SET POINT WRAPPING SPEED UPWARDS, CARRIAGE
   SET_POINT_HI_SPEED_CARR : INT  := 100;	//SET POINT HIGH SPEED, CARRIAGE
   TOP_PLATE : BOOL ;	//PROGRAMME LAY OUT TOP PLATE
   TOP_FILM : BOOL ;	//PROGRAMME LAY OUT TOP FILM
   WATERPROFE_TOP_FILM : BOOL ;	//PROGRAMME LAY OUT LOADCASSETTE
   FILMWELDING : BOOL ;	//PROGRAMME LAY OUT FILMWELDING
   HOT_AIR_FILMWELDING : BOOL ;	//PROGRAMME LAY OUT HOT AIR FILMWELDING
   SPARE_40 : INT ;
   SPARE_42 : INT ;
   SPARE_44 : INT ;
   CARR_STOP_AFTER_PC : INT  := 1;	//CARRIAGE STOP AFTER PHOTOCELL
   CARR_DOWN_BEFORE_CUT : INT ;	//CARRIAGE DOWN BEFORE CUTTING
   FILMWELDIND_TIME : S5TIME  := S5T#180MS;	//FILMWELDING TIME
   SET_POINT_CONT_BEFORE_HS : INT  := 24;	//SET POINT PULSES BEFORE HIGH SPEED
   SPARE_54 : INT ;
   SPARE_56 : INT ;
  END_STRUCT ;	
BEGIN
   PRG_CHOICE_OP3 := 1;
   PRG_POINTER := 1;
   FILMTENSION_TOP := 10;
   FILMTENSION_MIDDLE := 10;
   FILMTENSION_BOTTOM := 10;
   SET_POINT_TOPWRAP := 1;
   SET_POINT_BOTTOMWRAP := 2;
   SET_POINT_MS_TO_LS_TT := 66;
   SET_POINT_MID_SPEED_TT := 40;
   SET_POINT_HI_SPEED_TT := 55;
   SET_POINT_WRA_SPEED_DOWN := 35;
   SET_POINT_WRAPP_SPEED_UP := 35;
   SET_POINT_HI_SPEED_CARR := 100;
   CARR_STOP_AFTER_PC := 1;
   FILMWELDIND_TIME := S5T#180MS;
   SET_POINT_CONT_BEFORE_HS := 24;
END_DATA_BLOCK

DATA_BLOCK "PROG_9_DATA"	// DB 29
AUTHOR : LKA
NAME : MAINDATA
VERSION : 0.1
  STRUCT
   PRG_CHOICE_OP3 : INT  := 1;	//PROGRAMME CHOICE FROM OP3
   EXTERNAL_PROGRAMME : INT ;	//EXTERNAL PROGRAMME CHOICE
   OLD_PRG_POINTER : INT ;	//OLD PROGRAMME VALUE
   PRG_POINTER : INT  := 1;	//PROGRAMME WHICH PARAMETR IS TO BE CHANGED
   ACTUAL_PROGRAMME : INT ;	//AKTUELLT PROGRAM SOM ANVÄNDS I FILMCYKELN
   ACTUAL_PROGRAMME_JUMP : INT ;	//JUMP VALUE TO FC 21-29
   SPARE_12 : INT ;
   SPARE_14 : INT ;
   FILMTENSION_TOP : INT  := 10;	//SET POINT FILMTENSION TOP
   FILMTENSION_MIDDLE : INT  := 10;	//SET POINT FILMTENSION MIDDLE
   FILMTENSION_BOTTOM : INT  := 10;	//SET POINT FILMTENSION BOTTOM
   SET_POINT_TOPWRAP : INT  := 1;	//SET POINT NUMBER OF TOPWRAP
   SET_POINT_BOTTOMWRAP : INT  := 2;	//SET POINT NUMBER OF BOTTOMWRAP
   SET_POINT_MS_TO_LS_TT : INT  := 66;
   SET_POINT_MID_SPEED_TT : INT  := 40;	//SET POINT MEDDLE SPEED, TURNTABLE
   SET_POINT_HI_SPEED_TT : INT  := 55;	//SET POINT HIGH SPEED, TURNTABLE
   SET_POINT_WRA_SPEED_DOWN : INT  := 35;	//SET POINT WRAPPING SPEED DOWNWARDS, CARRIAGE
   SET_POINT_WRAPP_SPEED_UP : INT  := 35;	//SET POINT WRAPPING SPEED UPWARDS, CARRIAGE
   SET_POINT_HI_SPEED_CARR : INT  := 100;	//SET POINT HIGH SPEED, CARRIAGE
   TOP_PLATE : BOOL ;	//PROGRAMME LAY OUT TOP PLATE
   TOP_FILM : BOOL ;	//PROGRAMME LAY OUT TOP FILM
   WATERPROFE_TOP_FILM : BOOL ;	//PROGRAMME LAY OUT LOADCASSETTE
   FILMWELDING : BOOL ;	//PROGRAMME LAY OUT FILMWELDING
   HOT_AIR_FILMWELDING : BOOL ;	//PROGRAMME LAY OUT HOT AIR FILMWELDING
   SPARE_40 : INT ;
   SPARE_42 : INT ;
   SPARE_44 : INT ;
   CARR_STOP_AFTER_PC : INT  := 1;	//CARRIAGE STOP AFTER PHOTOCELL
   CARR_DOWN_BEFORE_CUT : INT ;	//CARRIAGE DOWN BEFORE CUTTING
   FILMWELDIND_TIME : S5TIME  := S5T#180MS;	//FILMWELDING TIME
   SET_POINT_CONT_BEFORE_HS : INT  := 24;	//SET POINT PULSES BEFORE HIGH SPEED
   SPARE_54 : INT ;
   SPARE_56 : INT ;
  END_STRUCT ;	
BEGIN
   PRG_CHOICE_OP3 := 1;
   PRG_POINTER := 1;
   FILMTENSION_TOP := 10;
   FILMTENSION_MIDDLE := 10;
   FILMTENSION_BOTTOM := 10;
   SET_POINT_TOPWRAP := 1;
   SET_POINT_BOTTOMWRAP := 2;
   SET_POINT_MS_TO_LS_TT := 66;
   SET_POINT_MID_SPEED_TT := 40;
   SET_POINT_HI_SPEED_TT := 55;
   SET_POINT_WRA_SPEED_DOWN := 35;
   SET_POINT_WRAPP_SPEED_UP := 35;
   SET_POINT_HI_SPEED_CARR := 100;
   CARR_STOP_AFTER_PC := 1;
   FILMWELDIND_TIME := S5T#180MS;
   SET_POINT_CONT_BEFORE_HS := 24;
END_DATA_BLOCK

DATA_BLOCK "INTERFACE_AREA"	// DB 30
AUTHOR : LKA
NAME : INTERF_A
VERSION : 0.1
  STRUCT
   OP3_CONTROLL_BITS_0 : BYTE ;
   OP3_CONTROLL_BITS_1 : BYTE ;
   OP3_CONTROLL_BITS_2 : BYTE ;
   OP3_RESERVED_1 : BYTE ;
   OP3_RESERVED_2 : BYTE ;
   OP3_RESERVED_3 : BYTE ;
   OP3_RESERVED_4 : BYTE ;
   OP3_RESERVED_5 : BYTE ;
   OP3_RESERVED_6 : BYTE ;
   OP3_RESERVED_7 : BYTE ;
   OP3_RESERVED_8 : BYTE ;
   OP3_RESERVED_9 : BYTE ;
   OP3_RESERVED_10 : BYTE ;
   OP3_CONNECTION_ID : BYTE ;
   OP3_RESERVED_11 : BYTE ;
   OP3_TIME_HOUR : BYTE ;
   OP3_TIME_MINUTE : BYTE ;
   OP3_TIME_SECOND : BYTE ;
   OP3_RESERVED_12 : BYTE ;
   OP3_RESERVED_13 : BYTE ;
   OP3_RESERVED_14 : BYTE ;
   OP3_DATE_DAY_OF_WEEK : BYTE ;
   OP3_DATE_DAY_OF_MONTH : BYTE ;
   OP3_DATE_MONTH : BYTE ;
   OP3_DATE_YEAR : BYTE ;
   OP3_RESERVED_15 : BYTE ;
   OP3_RESERVED_16 : BYTE ;
   OP3_RESERVED_17 : BYTE ;
   OP3_RESERVED_18 : BYTE ;
   OP3_RESERVED_19 : BYTE ;
   OP3_RESERVED_20 : BYTE ;
   OP3_RESERVED_21 : BYTE ;
   OP_SCREEN_NUMBER_READ : BYTE ;
   OP_ENTRY_NUMMBER_READ : BYTE ;
   OP_SCREEN_NUMBER_WRITE : BYTE ;
   OP_ENTRY_NUMMBER_WRITE : BYTE ;
   OP_SYSTEM_KEY_ASSIG : DWORD ;
  END_STRUCT ;	
BEGIN
   OP3_CONTROLL_BITS_0 := B#16#4;
   OP3_CONTROLL_BITS_1 := B#16#1;
   OP3_TIME_HOUR := B#16#15;
   OP3_TIME_MINUTE := B#16#24;
   OP3_DATE_DAY_OF_WEEK := B#16#3;
   OP3_DATE_DAY_OF_MONTH := B#16#8;
   OP3_DATE_MONTH := B#16#1;
   OP3_DATE_YEAR := B#16#2;
   OP_SCREEN_NUMBER_READ := B#16#8;
   OP_ENTRY_NUMMBER_READ := B#16#8;
   OP_SYSTEM_KEY_ASSIG := DW#16#8000;
END_DATA_BLOCK

DATA_BLOCK "MPI_GD"	// DB 100
VERSION : 0.1
  STRUCT
   IN : STRUCT
    Life_Bit_Szafa : BOOL ;
    Szafa_Automatyka : BOOL ;
    Foto_1_Banda_10 : BOOL ;
    Foto_2_Banda_10 : BOOL ;
    Foto_Banda_11 : BOOL ;
    Silnik_10_OK : BOOL ;
    Silnik_11_OK : BOOL ;
    Zabierz_Na_Bande_10 : BOOL ;
    Zezwolenie_Na_Wyjazd_11 : BOOL ;
    Potw_Dost_Na_Wyjazd_11 : BOOL ;
    Obrot_Na_Poz_Wlot_1 : BOOL ;
    Zmien_Program_Na_4 : BOOL ;
    Zmien_Pragram_Na_3 : BOOL ;
    Foto_Banda_9 : BOOL ;
    Help_INT : INT ;
   END_STRUCT ;
   OUT : STRUCT
    Life_Bit_Foliarka : BOOL ;
    Foliarka_Automatyka : BOOL ;
    Foliarka_Reczny : BOOL ;
    Foto_Banda_1 : BOOL ;
    Foto_Owijarka : BOOL ;
    Rezerwa_1 : BOOL ;
    Motor_10_Lewo : BOOL ;
    Motor_10_Prawo : BOOL ;
    Motor_11_Lewo : BOOL ;
    Motor_11_Prawo : BOOL ;
    Zezwolenie_Na_Wjazd_10 : BOOL ;
    Potw_Dost_Na_Wjazd_10 : BOOL ;
    Zabierz_Na_Bande_11 : BOOL ;
    Paleta_Obecna_Na_7_Tr : BOOL ;
    Paleta_Obraca_Sie : BOOL ;
    Foliowanie_Zakonczone : BOOL ;
    Banda_Fol_4_Foto_Tyl : BOOL ;
    Banda_Fol_4_Foto_Przod : BOOL ;
    Banda_Fol_4_Motor_Tyl : BOOL ;
    Banda_Fol_4_Motor_Przod : BOOL ;
    Bamda_Fol_Obr_Foto_Tyl : BOOL ;	//Wirtualna fotokomorka tylna banda obr
    Banda_Fol_Obr_Foto_Przod : BOOL ;	//Wirtualna fotokomorka przod banda obr
    Banda_Fol_Obr_Motor_Tyl : BOOL ;
    Banda_Fol_Obr_Motor_Przo : BOOL ;
    Banda_Fol_6_Foto_Tyl : BOOL ;
    Banda_Fol_6_Foto_Przod : BOOL ;
    Banda_Fol_6_Motor_Tyl : BOOL ;
    Banda_Fol_6_Motor_Przod : BOOL ;
   END_STRUCT ;
  END_STRUCT ;	
BEGIN
END_DATA_BLOCK

ORGANIZATION_BLOCK "MAIN_ORGANIZATION"	// OB 1
TITLE = MAIN ORGANIZATION
//                        Projekt :  01137855
//                                     
//                                                               
//  
//*************************************************************************
// Besteller            : Bauer Druck Nowogrodziec/Polen
// Maschinenbenennung   : GL1000 und Fördertechnik
// Kunde                : Bauer Druck Nowogrodziec(Polen)
//*************************************************************************
// Zeichnungsidentnr.   : *72017607*                                    
// Konstruktion         : Olc                                        
// Erstellungsdatum     : 30.10.2006                                    
//
//*************************************************************************
// Datum der Änderung   :   .  .               Name : . . . . . . .     
//                          .  .                      . . . . . . .     
//                          .  .                      . . . . . . .     
//
//*************************************************************************
// Steuerung            : SIMATIC S7 CPU 313C       
// Deckblatt            : Baustein OB1 Legende
// Software             : Siemens Step7 V5.4 SP1/ Protool Lite V 6.0 SP2
// MPI-Adressen         : nicht vernetzt
// Mittlere Zykluszeit  : ca. 9 ms
//*************************************************************************
//     MPI-Netzwerk:
//     Adresse:     Teilnehmer:
//     1       =    OP3
//     2       =    CPU
//     3       =    
//     4       =    
//     5       =    
//     6       =    
//*************************************************************************  
//
//Programmbausteine :
//     FC  1  Sammelmerker
//     FC  3  Bereichsabsicherung
//     FC  4  Lampentest
//     FC  5  Kundenmeldungen
//
//     FC 10  Betriebsarten
//     FC 11  Programmvorwahl  
//     FC 12  Motor Drehteller > Kupplung Roba 
//     FC 13  Grundstellungszyklus
//     FC 14  Transportzyklus
//     FC 15  Wickelzyklus
//     FC 16  Start nach 90Grad Einlauf
//     FC 17  90 Grad Einlauf
//     FC 18  90 Grad Auslauf
//     FC 19  Drehteller 0G.<>90G.
//     FC 21  Palettenpositionierung
//     FC 22  Drehteller
//     FC 23  Wickelschlitten
//     FC 24  Niederhalter
//     FC 25  Stretchsystem
//     FC 26  Folienklemmsystem
//     FC 27  Folie abschneiden
//     FC 28  Heissluft ansiegeln
//     FC 29  Kontaktschweissen
//     FC 32  Drehteller Positionszähler
//     FC 33  Wickelschlitten Positionszähler
//     FC 34  Allg. Zähler
//
//     FC 71  Förderer Pos.1
//     FC 72  Förderer Pos.2
//     FC 73  Förderer Pos.3
//     FC 74  Förderer Pos.4
//     FC 76  Förderer Pos.6
//     FC 77  Förderer Pos.7
//
//     FC110  Handling OP3
//     FC111  Betriebsart Hand
//     FC120  Aufbereitung Fehlermeldungen
//
//
//     OB  1  Programmorganisation/Legende
//
//     DB 12  Daten aktuelles Programm
//     DB 13  Daten Programmeditierung
//     DB 21  Daten Programm 1
//     DB 22  Daten Programm 2
//     DB 23  Daten Programm 3
//     DB 24  Daten Programm 4
//     DB 25  Daten Programm 5
//     DB 26  Daten Programm 6
//     DB 27  Daten Programm 7
//     DB 28  Daten Programm 8
//     DB 29  Daten Programm 9
//     DB 30  Schnittstelle OP3
//
AUTHOR : LKA
NAME : MAIN_CON
VERSION : 0.1
VAR_TEMP
  OB1_EV_CLASS : BYTE ;	//Bits 0-3 = 1 (Coming event), Bits 4-7 = 1 (Event class 1)
  OB1_SCAN_1 : BYTE ;	//1 (Cold restart scan 1 of OB 1), 3 (Scan 2-n of OB 1)
  OB1_PRIORITY : BYTE ;	//1 (Priority of 1 is lowest)
  OB1_OB_NUMBR : BYTE ;	//1 (Organization block 1, OB1)
  OB1_RESERVED_1 : BYTE ;	//Reserved for system
  OB1_RESERVED_2 : BYTE ;	//Reserved for system
  OB1_PREV_CYCLE : INT ;	//Cycle time of previous OB1 scan (milliseconds)
  OB1_MIN_CYCLE : INT ;	//Minimum cycle time of OB1 (milliseconds)
  OB1_MAX_CYCLE : INT ;	//Maximum cycle time of OB1 (milliseconds)
  OB1_DATE_TIME : DATE_AND_TIME ;	//Date and time OB1 started
END_VAR
BEGIN
NETWORK
TITLE = JUMP TO FC 1, CONTROL
      CALL  "CONTROL";
NETWORK
TITLE = PREVIOUS CYCLE TIME
      L     #OB1_PREV_CYCLE;
      T     "RUNNING_PROG".PREVCYCLETIME;
NETWORK
TITLE = MIN CYCLE TIME
      L     #OB1_MIN_CYCLE;
      L     "RUNNING_PROG".MINCYCLETIME;
      >I;
      JC    M001;
      L     #OB1_MIN_CYCLE;
      T     "RUNNING_PROG".MINCYCLETIME;
M001: NOP   0;
NETWORK
TITLE = RESET MIN CYCLE TIME
      AN    DB12.DBX 180.1;
      JC    M002;
      L     999;
      T     "RUNNING_PROG".MINCYCLETIME;
      R     DB12.DBX 180.1;
M002: NOP   0;
NETWORK
TITLE = MAX CYCLE TIME
      L     #OB1_PREV_CYCLE;
      L     "RUNNING_PROG".MAXCYCLETIME;
      <I;
      JC    M003;
      L     #OB1_PREV_CYCLE;
      T     "RUNNING_PROG".MAXCYCLETIME;
M003: NOP   0;
NETWORK
TITLE = RESET MAX CYCLE TIME
      AN    DB12.DBX 180.0;
      JC    M004;
      L     0;
      T     "RUNNING_PROG".MAXCYCLETIME;
      R     DB12.DBX 180.0;
M004: NOP   0;
END_ORGANIZATION_BLOCK

SYMBOL_TABLE
"AIO"	DB 10	DB 10
"Blok_Para"	DB 12	DB 12
"Blok_Bledow_Program"	DB 13	DB 13
"Asi_input_Transport"	DB 80	DB 80
"Asi_output_Transport"	DB 81	DB 81
"Asi_Input_Gender"	DB 82	DB 82
"Asi_Output_Gender"	DB 83	DB 83
"MPI_GD"	DB 100	DB 100	// Blok wymiany danych po mpi
"Blok_Bledow"	DB 119	DB 119
"DB_HMI"	DB 120	DB 120	// Blok wejsc wyjsc HMI
"Kom_Shuttle"	DB 205	DB 205
"Rejestr Band"	DB 310	DB 310
"Rejestr_Band_HMI"	DB 311	DB 311
"TEST_OBR2"	FB 2	FB 2	// Test obrotnicy nr 2
"Czesc_Bindujaca"	FB 3	FB 3	// Blok jazdy band bindownicy
"Czesc_Trasnportujaca"	FB 5	FB 5
"Filtr_zbocza_2"	FB 14	FB 14
"T_ON"	FB 20	FB 20	// Timer on delay with memory
"T_ON_+_RESET"	FB 21	FB 21	// Czasowka on delay z zapamietanym czasem  + reset
"Banda_Podwojna"	FB 29	FB 29
"Banda_Pojedyncza"	FB 30	FB 30
"Banda_Obr_1"	FB 31	FB 31	// Banda obrotowa o dwoch wlotach i jednej fotokomorce
"Banda_Obr_2"	FB 32	FB 32	// Banda obrotowa nr 2
"Banda_Poj_+Tryb_Reczny"	FB 33	FB 33
"Banda_Obr_Bind"	FB 34	FB 34	// Banda obrotowa sluzaca do bindowania
"Blok_Pracy_Bindownicy"	FB 35	FB 35	// funkcja pozycjonujaca bande
"Wybranie_Wjazdu"	FB 50	FB 50
"Obr_Na_Poz_1"	FB 51	FB 51
"Obr_Na_Poz_2"	FB 52	FB 52	// Obrot na pozycje uwzgledniajacy czujniki 45st
"Obr_Na_Poz_3"	FB 53	FB 53	// Funkcja sterujaca obrotem talerza 4 po³o¿enia.
"Obr_Na_Poz_4"	FB 54	FB 54
"Pozycjonowanie_Bandy"	FB 55	FB 55
"Poz_Band_Back"	FB 56	FB 56
"Bindownica_Test"	FB 57	FB 57	// Testowy blok wejsc wyjsc bindownicy
"Pozycjonowanie_Palety"	FB 58	FB 58	// Funkcja pozycjonujaca palete
"TSEND"	FB 63	FB 63	// Send Data
"TRCV"	FB 64	FB 64	// Receive Data
"Blok_kodow_Pracy"	FB 80	FB 80
"Funkcja_Bezp_Transport"	FC 2	FC 2
"Funkcja_Bezp_Gender"	FC 3	FC 3
"Sprawdzenie_Czujnikow"	FC 4	FC 4
"Szukaj_Zmiany"	FC 5	FC 5	// Funkcja szukajaca zmiany w obszarze odwzorowania
"FC_Lampki"	FC 6	FC 6	// Funkcja sterujaca lampkami
"Szukaj_Zmiany_2"	FC 7	FC 7
"Toggle"	FC 8	FC 8	// Funkcja przycisku bistabilnego
"Sterwanie_Swiatlo"	FC 9	FC 9	// Sterowanie sygnalami swietlnymi
"Lampka_Blad"	FC 10	FC 10
"Przyciski_Dwufunkcyjne"	FC 11	FC 11
"Przyporzadkowanie_Wejsc"	FC 20	FC 20
"Przyporzadkowanie_Wyjsc"	FC 21	FC 21
"Przyp_Wejsc_Gender"	FC 22	FC 22
"Przyp_Wysc_Gender"	FC 23	FC 23
"Rejestr_Tasm"	FC 30	FC 30
"FC_Auto_Reczny"	FC 40	FC 40
"Przycisk_Reset"	FC 41	FC 41	// Kasowanie_Bledow
"Wybor_Wjazdu"	FC 50	FC 50	// Wybor miejsca pobierania palety
"Obrotnica_Na_Pozycje"	FC 51	FC 51
"ASI_Odczyt"	FC 80	FC 80
"ASI_Zapis"	FC 81	FC 81
"Opoznienie_Wylotu"	FC 85	FC 85
"Opoznienie_Wlotu"	FC 86	FC 86	// Funkcja opozniajaca wlot
"Opoznienie_Wlotu_2"	FC 87	FC 87
"Komunikacja_GD"	FC 100	FC 100	// Komunikacja szafa foliarka
"Obsluga bledow"	FC 119	FC 119	// funkcja przekazujaca bledy do bloku db
"FC_HMI"	FC 120	FC 120
"Step_Control"	FC 127	FC 127	// Kontrola krokow
"Inkrementacja_Kroku"	FC 128	FC 128	// Funkcja inkrementujaca kroku
"Step_Control_2"	FC 130	FC 130
"Utworz_Blad"	FC 132	FC 132	// Funkcja stwarz kod bledu
"Funkcja_Zegara"	FC 140	FC 140	// Funkcja zegara
"Komunikacja_Gender"	FC 205	FC 205
"Monitor_Band_Lini"	FC 310	FC 310
"Monitor_Bandy"	FC 313	FC 313	// Funkcja monitorujaca przejezdzajacy produkt
"Monitor_Bandy_Obr"	FC 314	FC 314
"Monitor_Bandy_+_Reczny"	FC 315	FC 315	// Funkcja monitorujaca + tryb reczny
"Monitor_Palety"	FC 316	FC 316	// Auto wyszukiwanie palety w masce
"Monitor_Bandy_2"	FC 317	FC 317	// Monitor Bandy z wykryciem auto
"Monitor_Bandy_Obr_2"	FC 318	FC 318
"Dekoduj_Maske"	FC 320	FC 320
"Nadpisz_Maske"	FC 321	FC 321
"Wirtualna_Foliarka"	FC 330	FC 330
"pb_Strefa_bezpieczenstwa"	I 0.0	BOOL
"pb_Reczny"	I 0.1	BOOL
"pb_Auto"	I 0.2	BOOL
"pb_Reset"	I 0.3	BOOL
"pb_Stop"	I 0.4	BOOL
"pb_Cykl_Start"	I 0.5	BOOL
"pb_Wozek_Tyl"	I 0.6	BOOL
"pb_Wozek_Przod"	I 0.7	BOOL
"pb_Tasma_1_Tyl"	I 1.0	BOOL
"pb_Tasma_1_Przod"	I 1.1	BOOL
"pb_Tasma_2_Tyl"	I 1.2	BOOL
"pb_Tasma_2_Przod"	I 1.3	BOOL
"pb_Tasma_Obr_Tyl"	I 1.4	BOOL
"pb_Tasma_Obr_Przod"	I 1.5	BOOL
"pb_Tasma_Wylot_Przod"	I 1.6	BOOL
"pb_Tasma_Wylot_Tyl"	I 1.7	BOOL
"Obwod_Bezp_Bindownicy"	I 2.0	BOOL
"Bind_Polozenie_Podst"	I 2.1	BOOL
"Blad_Bindownicy"	I 2.2	BOOL
"Start_Koniec_Wiazania"	I 2.3	BOOL
"Bindownica_Auto"	I 2.4	BOOL	// Bindownica jest w trybie automatyki
"rez_i_2_5"	I 2.5	BOOL
"Prasa_W_Gorze"	I 2.6	BOOL
"Foto_Wozek"	I 2.7	BOOL
"i_foto_lewo_1"	I 3.0	BOOL
"i_foto_lewo_2"	I 3.1	BOOL
"i_foto_prawo_1"	I 3.2	BOOL
"i_foto_prawo_2"	I 3.3	BOOL
"PB_Funkcja"	I 3.4	BOOL
"Przek_Bezp_Gender_OK"	I 3.5	BOOL
"Przekaznik_Kurtyn_OK"	I 3.6	BOOL
"rez_i_3_7"	I 3.7	BOOL
"Przekaznik_Bezp_OK"	I 4.0	BOOL
"Start"	I 4.1	BOOL
"Stop"	I 4.2	BOOL
"Praca_Z_Etykietami"	I 4.3	BOOL
"Przek_Rejonu_Bind_Ok"	I 4.4	BOOL	// Uwaga wycinanie
"Silownik_Etyk_Tyl"	I 5.0	BOOL
"Etyk_Gotowa"	I 5.1	BOOL
"Dane_W_Drukarce"	I 5.2	BOOL
"Brak_Papieru"	I 5.3	BOOL
"Drukuj_Recznie"	I 5.4	BOOL
"Bity_Przyciskow"	IB 0	BYTE
"Wejscia_Shuttle_1"	ID 68	DWORD
"Wejscia_Shuttle_2"	ID 72	DINT
"Zawsze_True"	M 0.0	BOOL
"Zawsze_False"	M 0.1	BOOL
"Marka_X"	M 0.3	BOOL	// Marka output wszystko jedno
"Help_Start"	M 1.0	BOOL
"Help_Zbocze_Start"	M 1.1	BOOL
"Help_Start_2"	M 1.2	BOOL
"Marka_Bezp_Transportera"	M 2.0	BOOL
"Marka_Start_Stop"	M 2.1	BOOL
"Marka_Bezpieczenstwa_2"	M 2.2	BOOL
"Rejon_Bindownicy_Stop"	M 2.3	BOOL
"Strefa_Bind_Ok"	M 2.4	BOOL
"Help_PB_Stop"	M 2.5	BOOL
"Gender_Wszystko_OK"	M 2.6	BOOL
"Freeze"	M 2.7	BOOL
"Brak_Bledu"	M 3.0	BOOL
"Falowniki_OK"	M 3.1	BOOL
"Fuse_OK"	M 3.2	BOOL
"Help_Freeze"	M 3.3	BOOL
"Marka_Bezpieczenstwa_3"	M 3.4	BOOL
"Zezwolenie_Na_Wjazd"	M 3.5	BOOL	// Do stawiania lini
"Stop_Hmi"	M 3.7	BOOL
"Not_Aus_27_OK"	M 4.0	BOOL
"Not_Aus_28_OK"	M 4.1	BOOL
"Not_Aus_29_OK"	M 4.2	BOOL
"Strefa_Bind_Zamk"	M 4.3	BOOL
"Not_Aus_30_OK"	M 4.4	BOOL
"Not_Aus_31_OK"	M 4.5	BOOL
"Zmiana_Wykryta"	M 5.0	BOOL
"Help_M5.1"	M 5.1	BOOL
"Cykl_Binowania_Przwyr"	M 5.2	BOOL
"Help_M5.3"	M 5.3	BOOL
"Help_M5.4"	M 5.4	BOOL
"Kat_Jazdy_Rolek_OK"	M 5.5	BOOL
"Kat_Obrotnicy_Bezp"	M 5.6	BOOL
"Kurtyny_Wlot_Ok"	M 6.0	BOOL
"Kurtyny_Wylot_Ok"	M 6.1	BOOL
"Rygiel_OK"	M 6.2	BOOL
"Wirt_Syg_Bezp_Gender"	M 6.3	BOOL
"M_Zez_Na_Prace_Bind"	M 6.4	BOOL
"M_Obwod_Bezp_Bind"	M 6.5	BOOL
"Help_M6.6"	M 6.6	BOOL
"Warunki_Startu_OK"	M 7.0	BOOL
"Help_Bit_M_7_1"	M 7.1	BOOL
"Edge_7.6"	M 7.6	BOOL
"Pomoc_Reczny"	M 7.7	BOOL
"M_Blad_Cyklu_Bindowania"	M 8.0	BOOL	// Blad cyklu
"M_Trick"	M 8.1	BOOL
"M_Cykl_Bindowania_Trwa"	M 9.0	BOOL
"Marka_Bezp_Gendera"	M 10.0	BOOL
"Falowniki_Gender_OK"	M 10.1	BOOL
"Edge_M11.0"	M 11.0	BOOL
"Edge_M11.1"	M 11.1	BOOL
"M_Reset_Bledow"	M 20.0	BOOL
"M_Reset_Krokow"	M 20.1	BOOL
"Help_M20.2"	M 20.2	BOOL
"M_Help_Reset_Bledow"	M 20.3	BOOL
"M_pb_Cykl_Start"	M 20.5	BOOL
"Auto_Sprawdzone"	M 20.6	BOOL
"M_Powrot_do_Stopu"	M 20.7	BOOL
"Brak_Bledow_Do_Auto"	M 21.0	BOOL	// Brak bledow przy pojsicu w auto
"Blad_Automatu"	M 21.1	BOOL	// Blad automatu
"Help_M21.2"	M 21.2	BOOL
"help_m21.3"	M 21.3	BOOL
"Edge_M22.0"	M 22.0	BOOL
"M_Foto_1_Banda_11"	M 30.0	BOOL
"M_Foto_1_Banda_14"	M 40.0	BOOL
"Help_M_40_1"	M 40.1	BOOL
"M_Foto_1_Tasma_1"	M 40.2	BOOL
"Help_M_40_3"	M 40.3	BOOL
"M_Foto_1_Banda_3"	M 40.4	BOOL
"Help_M_40_5"	M 40.5	BOOL
"M_Foto_1_Banda_12"	M 40.6	BOOL
"Help_M_40_7"	M 40.7	BOOL
"Help_Foto"	M 41.0	BOOL
"M_Foto_1_Banda_2"	M 41.1	BOOL
"Zboczne_M44.0"	M 44.0	BOOL
"M_Wypchnie_Palety"	M 44.1	BOOL
"Woz_Zez_R_Do_Nast"	M 45.0	BOOL
"Zabierz_Palete_Wozek"	M 45.1	BOOL
"Bini_Prasa_Pol_Podst"	M 50.0	BOOL
"M_Bindownica_Poz_Podst"	M 50.1	BOOL
"M_Foto_1_Opoz"	M 90.0	BOOL	// Opoznienie fotokomorki dla Gender onlline
"Auto_Reczny"	M 120.0	BOOL	// auto-1;reczny 0
"Auto_Reczny_3"	M 120.1	BOOL
"PB_Stop_Panel"	M 120.3	BOOL
"Test_Lamp"	M 121.0	BOOL
"Help_Lam_Czerwona"	M 122.0	BOOL
"Help_Lam_Strzal_Tas"	M 122.1	BOOL
"Help_Lam_pb_strefa"	M 122.2	BOOL
"Help_Lam_pb_reczny"	M 122.3	BOOL
"Help_Lam_pb_auto"	M 122.4	BOOL
"Help_Lam_pb_reset"	M 122.5	BOOL
"Help_lam_pb_stop"	M 122.6	BOOL
"Help_Lam_pb_start"	M 122.7	BOOL
"Help_M123.0"	M 123.0	BOOL
"Help_Lam_Biala"	M 123.1	BOOL
"Help_Lam_Blad_Lini"	M 123.2	BOOL
"Help_Lamp_Zielona"	M 123.3	BOOL
"M_PB_Lampka_Obr"	M 123.4	BOOL
"M_Lampka_PB_Funkcja"	M 123.5	BOOL
"VPB_Tyl_Tasma_3_Tyl"	M 124.0	BOOL
"VPB_Tasma_3_Przod"	M 124.1	BOOL
"VPB_Obrot_CW"	M 124.2	BOOL
"VPB_Obrot_CCW"	M 124.3	BOOL
"Help_M182.2"	M 180.2	BOOL
"Help_M180.3"	M 180.3	BOOL
"Komunikacja_OK"	M 181.0	BOOL
"M_Miganie_200ms"	M 200.0	BOOL
"M_Miganie_500ms"	M 200.1	BOOL
"M_Miganie_100ms"	M 200.2	BOOL
"BA_Bindownica_Nie_Podst"	M 210.0	BOOL
"Bindownica_Brak_Bezp"	M 210.1	BOOL
"Blad_Foto_Tasma_1"	M 210.2	BOOL
"Blad_Foro_Tasma_2"	M 210.3	BOOL
"Blad_Foto_Tasma_4"	M 210.4	BOOL
"M_Binownica_Blad"	M 210.5	BOOL
"Blad_Fotokomorek_Obr"	M 210.6	BOOL
"Obr_Nie_W_Pozycji"	M 210.7	BOOL
"Blad_Kom_Wozke"	M 300.0	BOOL
"Wym_Online_Gender"	M 300.1	BOOL
"Wym_OFFline_Gender"	M 300.2	BOOL	// Wymuszenie z odbierania
"Edge_300.3"	M 300.3	BOOL
"Edge_M300.4"	M 300.4	BOOL
"Linia_Gender_ONline"	M 310.0	BOOL
"ON_Wiazanie_Poprzeczne"	M 602.0	BOOL
"ON_Wiazanie_Wzdluzne"	M 602.1	BOOL
"ON_Deklowanie"	M 602.2	BOOL
"Wybrane_Foliowanie"	M 602.4	BOOL
"Foliowanie_Zawsze"	M 602.5	BOOL
"ON_2_Poprzeczne"	M 603.0	BOOL
"ON_2_Wzdluzne"	M 603.1	BOOL
"ON_2_Deklowanie"	M 603.2	BOOL
"Info_Koniec_Cyklu"	M 604.0	BOOL
"Edge_M604.1"	M 604.1	BOOL
"Zbocze_M604.5"	M 604.5	BOOL
"Nadpisz_Foliarke"	M 604.6	BOOL
"Masz_Info_Bit_0"	M 605.0	BOOL
"Masz_Info_Bit_1"	M 605.1	BOOL
"Masz_Info_Bit_2"	M 605.2	BOOL
"Masz_Info_Bit_3"	M 605.3	BOOL
"Byte_Bledu"	MB 10	BYTE
"Nowe_Slowo"	MD 20	DWORD
"Stare_Slowo"	MD 24	DWORD
"Nowe_Slowo_1"	MD 400	DWORD
"Stare_Slowo_1"	MD 404	DWORD
"Nowe_Slowo_2"	MD 408	DWORD
"Stare_Slowo_2"	MD 412	DWORD
"Nowe_Slowo_do_Freeze"	MD 416	DWORD
"Stare_Slowo_do_Freeze"	MD 420	DWORD
"Help_MW12"	MW 12	WORD
"Help_MW14"	MW 14	INT
"Help_MW16"	MW 16	S5TIME
"Help_MW_30"	MW 30	INT
"Help_MW620"	MW 620	WORD
"Help_MW622"	MW 622	WORD
"Help_MW624"	MW 624	WORD
"Help_MW626"	MW 626	WORD
"Help_MW628"	MW 628	WORD
"Help_MW630"	MW 630	WORD
"Help_MW632"	MW 632	WORD
"Help_MW634"	MW 634	WORD
"Help_MW636"	MW 636	WORD
"Help_MW638"	MW 638	WORD
"Help_MW640"	MW 640	WORD
"Help_MW642"	MW 642	WORD
"Help_MW644"	MW 644	WORD
"Help_MW646"	MW 646	WORD
"Help_MW648"	MW 648	WORD
"Help_MW650"	MW 650	WORD
"Help_MW652"	MW 652	WORD
"Help_MW654"	MW 654	WORD
"Help_MW656"	MW 656	WORD
"Help_MW658"	MW 658	WORD
"I/O_FLT1"	OB 82	OB 82	// I/O Point Fault 1
"RACK_FLT"	OB 86	OB 86	// Loss of Rack Fault
"COMPLETE RESTART"	OB 100	OB 100	// Complete Restart
"PROG_ERR"	OB 121	OB 121	// Programming Error
"MOD_ERR"	OB 122	OB 122	// Module Access Error
"Lampka_Blad_Bind"	Q 0.0	BOOL
"Lampka_PB_Funkcja"	Q 0.1	BOOL
"Lampka_pb_Strefa_Bezp"	Q 0.2	BOOL
"Lampka_pb_Reczny"	Q 0.3	BOOL
"Lampka_pb_Auto"	Q 0.4	BOOL
"Lampka_pb_Reset"	Q 0.5	BOOL
"Lampka_pb_Stop"	Q 0.6	BOOL
"Lampka_pb_Cykl_Start"	Q 0.7	BOOL
"Zawor_Prasa"	Q 1.0	BOOL
"Zezw_na_prace_Bind"	Q 1.1	BOOL
"o_Start_Wiazania"	Q 1.2	BOOL
"rez_q_1_3"	Q 1.3	BOOL
"PB_Lampka_Obr"	Q 1.4	BOOL
"rez_q_1_5"	Q 1.5	BOOL
"Lampka_Lewo_Ok"	Q 1.6	BOOL
"Lampka_Prawo_Ok"	Q 1.7	BOOL
"Reset_Przek_Bezp_Gen_1"	Q 2.0	BOOL	// Reset przekaznika bezpieczenstwa od Gender not-aus
"Reset_Przek_Bezp_Gen_2"	Q 2.1	BOOL
"Lampka_Strzal"	Q 2.2	BOOL
"Reset_P_Bezp"	Q 8.0	BOOL
"Lampka_Biala"	Q 8.1	BOOL
"Lampka_Blad_Lini"	Q 8.2	BOOL
"Lampa_Zielona"	Q 8.3	BOOL
"Silownik_Etykiet"	Q 8.4	BOOL
"Drukuj_Etykiete"	Q 8.5	BOOL
"Zalacz_Skaner"	Q 8.6	BOOL
"Rezerwa_Q_4_7"	Q 8.7	BOOL
"Lampka_Obraz_W_Pamieci"	Q 9.0	BOOL
"Reset_P_Bepz_Strefa"	Q 9.1	BOOL
"Wyjscia_Do_Shuttle"	QD 60	DWORD
"Wyjscia_Do_Shuttle_2"	QD 64	DINT
"TON"	SFB 4	SFB 4	// Generate an On Delay
"READ_CLK"	SFC 1	SFC 1	// Read System Clock
"WR_REC"	SFC 58	SFC 58	// Write Data Record
"RD_REC"	SFC 59	SFC 59	// Read a Data Record
"Help_T5"	T 5	TIMER
"Timmer_T32"	T 12	TIMER
"T30_Test_Lampek"	T 30	TIMER
"Auto_Ghost_Mode"	T 37	TIMER
"T50_Monitoring"	T 50	TIMER
"T51_Monitoring"	T 51	TIMER
"T52_Monitoring"	T 52	TIMER
"T53_Monitoring"	T 53	TIMER
"T54_Monitoring"	T 54	TIMER
"Help_T55"	T 55	TIMER
"Help_T56"	T 56	TIMER
"Help_T57"	T 57	TIMER
"Help_T58"	T 58	TIMER
"Help_T59"	T 59	TIMER
"Help_T60"	T 60	TIMER
"Help_T61"	T 61	TIMER
"Help_T62"	T 62	TIMER
"Help_T63"	T 63	TIMER
"Help_T64"	T 64	TIMER
"Help_T65"	T 65	TIMER
"Help_T66"	T 66	TIMER
"Help_T67"	T 67	TIMER
"Help_T68"	T 68	TIMER
"Help_T69"	T 69	TIMER
"Help_T70"	T 70	TIMER
"Help_T71"	T 71	TIMER
"T90"	T 90	TIMER
"T91"	T 91	TIMER
"Timmer_T100"	T 100	TIMER
"SEW_Model"	UDT 1	UDT 1	// Model SEW'a
"CROSS_Model"	UDT 2	UDT 2
"ESTOP_Model"	UDT 3	UDT 3
"BRAMA_Model"	UDT 4	UDT 4
"PB_Model"	UDT 5	UDT 5	// Model przycisku
"OBROTOWA_Model"	UDT 6	UDT 6	// Model sygnalow z bandy obrotowej
"CZUJNIKI_1_Model"	UDT 7	UDT 7	// Model czujnikow na obrotnicy
"CZUJNIKI_2_Model"	UDT 8	UDT 8
"S_Model"	UDT 9	UDT 9
"CZUJNIKI_3_MODEL"	UDT 10	UDT 10
"OBROTOWA_2_MODEL"	UDT 11	UDT 11
"RESET_MODEL"	UDT 12	UDT 12
"Wzor_Pracy"	UDT 20	UDT 20
"VAT_1"	VAT 1	
"VAT_1g"	VAT 2	
"VAT_Para"	VAT 5	
"VAT_Monitor"	VAT 6	
END_SYMBOL_TABLE

TYPE "SEW_Model"	// UDT 1
VERSION : 0.1
  STRUCT
   Silnik_OK : BOOL ;	//Silnik ok
   Rezerwa_Silnik : BOOL ;
   Foto_1 : BOOL ;	//Wejscie SEW 1
   Foto_2 : BOOL ;	//Wejscie SEW 2
   C_Wise : BOOL ;	//ClockWise
   CC_Wise : BOOL ;	//CounterClockWise
   Wolno : BOOL ;	//Wolno
   S_Bit : BOOL ;	//Bit bezpieczenstwa
   Zez_Do_Pop : BOOL ;	//Zezwolenie do poprzedniej
   Paleta_Dost_do_Pop : BOOL ;	//Potwierdzenie dostarczenia
   Zabierz_do_Nast : BOOL ;	//Przejecie palety do nast
   Paleta_Poprawna : BOOL ;	//Wykorzystywane do monitoringu
   Res_1_4 : BOOL ;
   Res_1_5 : BOOL ;
   Zez_Reczny_do_Pop : BOOL ;	//Zezwolenie na reczny tyl
   Zez_Reczny_do_Nast : BOOL ;	//Zezwolenie na reczny przod
  END_STRUCT ;	
END_TYPE

TYPE "CROSS_Model"	// UDT 2
VERSION : 0.1
  STRUCT
   OSSD_Tor_1_1 : BOOL ;
   OSSD_Tor_1_2 : BOOL ;
   OSSD_Tor_2_1 : BOOL ;
   OSSD_Tor_2_2 : BOOL ;
   Rez_0_4 : BOOL ;
   Rez_0_5 : BOOL ;
   Rez_0_6 : BOOL ;
   Rez_0_7 : BOOL ;
   Rez_1_0 : BOOL ;
   Rez_1_1 : BOOL ;
   Rez_1_2 : BOOL ;
   Rez_1_3 : BOOL ;
   Rez_1_4 : BOOL ;
   Rez_1_5 : BOOL ;
   Rez_1_6 : BOOL ;
   Rez_1_7 : BOOL ;
  END_STRUCT ;	
END_TYPE

TYPE "ESTOP_Model"	// UDT 3
VERSION : 0.1
  STRUCT
   EStop_Tor_1_1 : BOOL ;
   EStop_Tor_1_2 : BOOL ;
   EStop_Tor_2_1 : BOOL ;
   EStop_Tor_2_2 : BOOL ;
   Rez_0_4 : BOOL ;
   Rez_0_5 : BOOL ;
   Rez_0_6 : BOOL ;
   Rez_0_7 : BOOL ;
   Rez_1_0 : BOOL ;
   Rez_1_1 : BOOL ;
   Rez_1_2 : BOOL ;
   Rez_1_3 : BOOL ;
   Rez_1_4 : BOOL ;
   Rez_1_5 : BOOL ;
   Rez_1_6 : BOOL ;
   Rez_1_7 : BOOL ;
  END_STRUCT ;	
END_TYPE

TYPE "PB_Model"	// UDT 5
VERSION : 0.1
  STRUCT
   Przycisk_Start : BOOL ;	//Start i reset ob. bezp
   Czujnik_Kolizji : BOOL ;
   Rez_0_2 : BOOL ;
   Rez_0_3 : BOOL ;
   Rez_0_4 : BOOL ;
   Rez_0_5 : BOOL ;
   Rez_0_6 : BOOL ;
   Rez_0_7 : BOOL ;
   Rez_1_0 : BOOL ;
   Rez_1_1 : BOOL ;
   Rez_1_2 : BOOL ;
   Rez_1_3 : BOOL ;
   Rez_1_4 : BOOL ;
   Rez_1_5 : BOOL ;
   Rez_1_6 : BOOL ;
   Rez_1_7 : BOOL ;
  END_STRUCT ;	
END_TYPE

TYPE "OBROTOWA_Model"	// UDT 6
VERSION : 0.1
  STRUCT
   Silnik_OK : BOOL ;	//Silnik ok
   Rezerwa_Silnik : BOOL ;
   Foto_1 : BOOL ;	//Wejscie SEW 1
   Foto_2 : BOOL ;	//Wejscie SEW 2
   C_Wise : BOOL ;	//ClockWise
   CC_Wise : BOOL ;	//CounterClockWise
   Wolno : BOOL ;	//Wolno
   S_Bit : BOOL ;	//Bit bezpieczenstwa
   Zez_Do_Pop_Wlot_1 : BOOL ;	//Zezwolenie do poprzedniej
   Potw_Dost_Wlot_1 : BOOL ;	//Potwierdzenie dostarczenia
   Zez_Do_Pop_Wlot_2 : BOOL ;	//Wykorzystywane do monitoringu
   Potw_Dost_Wlot_2 : BOOL ;
   Przejmij_Palete : BOOL ;	//Przejecie palety do nast
   Rez_1_6 : BOOL ;
   Paleta_Poprawna_1 : BOOL ;	//Wykorzystywane do monitoringu
  END_STRUCT ;	
END_TYPE

TYPE "CZUJNIKI_1_Model"	// UDT 7
VERSION : 0.1
  STRUCT
   Czujnik_0_St : BOOL ;
   Czujnik_Ham_0_St : BOOL ;
   Czujnik_Ham_90_St : BOOL ;
   Czujnik_90_St : BOOL ;
   Rez_0_4 : BOOL ;
   Rez_0_5 : BOOL ;
   Rez_0_6 : BOOL ;
   Rez_0_7 : BOOL ;
   Rez_1_0 : BOOL ;
   Rez_1_1 : BOOL ;
   Rez_1_2 : BOOL ;
   Rez_1_3 : BOOL ;
   Rez_1_4 : BOOL ;
   Rez_1_5 : BOOL ;
   Rez_1_6 : BOOL ;
   Rez_1_7 : BOOL ;
  END_STRUCT ;	
END_TYPE

TYPE "CZUJNIKI_2_Model"	// UDT 8
VERSION : 0.1
  STRUCT
   Czujnik_45_St_CW : BOOL ;
   Czujnik_45_St_CCW : BOOL ;
   Rez_0_2 : BOOL ;
   Rez_0_3 : BOOL ;
   Rez_0_4 : BOOL ;
   Rez_0_5 : BOOL ;
   Rez_0_6 : BOOL ;
   Rez_0_7 : BOOL ;
   Rez_1_0 : BOOL ;
   Rez_1_1 : BOOL ;
   Rez_1_2 : BOOL ;
   Rez_1_3 : BOOL ;
   Rez_1_4 : BOOL ;
   Rez_1_5 : BOOL ;
   Rez_1_6 : BOOL ;
   Rez_1_7 : BOOL ;
  END_STRUCT ;	
END_TYPE

TYPE "S_Model"	// UDT 9
VERSION : 0.1
  STRUCT
   Silnik_OK : BOOL ;	//Silnik ok
   Rezerwa_Silnik : BOOL ;
   Foto_1 : BOOL ;	//Wejscie SEW 1
   Foto_2 : BOOL ;	//Wejscie SEW 2
   C_Wise : BOOL ;	//ClockWise
   CC_Wise : BOOL ;	//CounterClockWise
   Wolno : BOOL ;	//Wolno
   S_Bit : BOOL ;	//Bit bezpieczenstwa
   Zez_Do_Pop_Wlot_1 : BOOL ;	//Zezwolenie do poprzedniej
   Potw_Dost_Wlot_1 : BOOL ;	//Potwierdzenie dostarczenia
   Zez_Do_Pop_Wlot_2 : BOOL ;	//Wykorzystywane do monitoringu
   Potw_Dost_Wlot_2 : BOOL ;
   Przejmij_Palete : BOOL ;	//Przejecie palety do nast
   Rez_1_6 : BOOL ;
   Paleta_Poprawna_1 : BOOL ;	//Wykorzystywane do monitoringu
  END_STRUCT ;	
END_TYPE

TYPE "CZUJNIKI_3_MODEL"	// UDT 10
VERSION : 0.1
  STRUCT
   Czujnik_Ham_180_St : BOOL ;
   Czujnik_180_St : BOOL ;
   Czujnik_Ham_270_St : BOOL ;
   Czujnik_270_St : BOOL ;
   Rez_0_4 : BOOL ;
   Rez_0_5 : BOOL ;
   Rez_0_6 : BOOL ;
   Rez_0_7 : BOOL ;
   Rez_1_0 : BOOL ;
   Rez_1_1 : BOOL ;
   Rez_1_2 : BOOL ;
   Rez_1_3 : BOOL ;
   Rez_1_4 : BOOL ;
   Rez_1_5 : BOOL ;
   Rez_1_6 : BOOL ;
   Rez_1_7 : BOOL ;
  END_STRUCT ;	
END_TYPE

TYPE "OBROTOWA_2_MODEL"	// UDT 11
VERSION : 0.1
  STRUCT
   Silnik_OK : BOOL ;	//Silnik ok
   Rezerwa_Silnik : BOOL ;
   Foto_1 : BOOL ;	//Wejscie SEW 1
   Foto_2 : BOOL ;	//Wejscie SEW 2
   C_Wise : BOOL ;	//ClockWise
   CC_Wise : BOOL ;	//CounterClockWise
   Wolno : BOOL ;	//Wolno
   S_Bit : BOOL ;	//Bit bezpieczenstwa
   Res_1_0 : BOOL ;	//Zezwolenie do poprzedniej
   Res_1_1 : BOOL ;	//Potwierdzenie dostarczenia
   Res_1_2 : BOOL ;	//Potwierdzenie dostarczenia
   Res_1_3 : BOOL ;	//Potwierdzenie dostarczenia
   Res_1_4 : BOOL ;	//Potwierdzenie dostarczenia
   Res_1_5 : BOOL ;	//Potwierdzenie dostarczenia
   Res_1_6 : BOOL ;	//Potwierdzenie dostarczenia
   Res_1_7 : BOOL ;	//Potwierdzenie dostarczenia
  END_STRUCT ;	
END_TYPE

TYPE "RESET_MODEL"	// UDT 12
VERSION : 0.1
  STRUCT
   Reset_Wlot : BOOL ;
   Reset_Wylot : BOOL ;
   RES_0_2 : BOOL ;
   RES_0_3 : BOOL ;
   Rez_0_4 : BOOL ;
   Rez_0_5 : BOOL ;
   Rez_0_6 : BOOL ;
   Rez_0_7 : BOOL ;
   Rez_1_0 : BOOL ;
   Rez_1_1 : BOOL ;
   Rez_1_2 : BOOL ;
   Rez_1_3 : BOOL ;
   Rez_1_4 : BOOL ;
   Rez_1_5 : BOOL ;
   Rez_1_6 : BOOL ;
   Rez_1_7 : BOOL ;
  END_STRUCT ;	
END_TYPE

TYPE "Wzor_Pracy"	// UDT 20
VERSION : 0.1
  STRUCT
   wiazanie_poprzeczne : BOOL ;
   wiazanie_wzdluzne : BOOL ;
  END_STRUCT ;	
END_TYPE

FUNCTION_BLOCK "Czesc_Bindujaca"	// FB 3
//Funkcja odpowiada za sterowanie lini bindujacej
//Uwzgledniony zostal tryb reczny
//
VERSION : 0.1
VAR
  Tasma_1 : FB 33;	//Adres 23
  Tasma_2 : FB 33;	//Adres 24
  Tasma_Obr_3 : FB 34;	//Adres 1 i 15
  Tasma_4 : FB 33;	//Adres 2
  Bin_IN_OUT : FB 57;
  Bind_Obwod_Ok : BOOL ;
  Bind_Poz_Podst : BOOL ;
  Bind_Sygn_Got : BOOL ;
  Bind_Blad : BOOL ;
  Bind_Start_Kon : BOOL ;
  Zaj_Nieb_2 : BOOL ;
  Zaj_Nieb_4 : BOOL ;
  Tasma_Rezerwa_1 : FB 33;
  Tasma_Rezerwa_2 : FB 33;
END_VAR
VAR_TEMP
  Temp_Bit_1 : BOOL ;
END_VAR
BEGIN
NETWORK
TITLE =
//Ten network celowo jest wolny
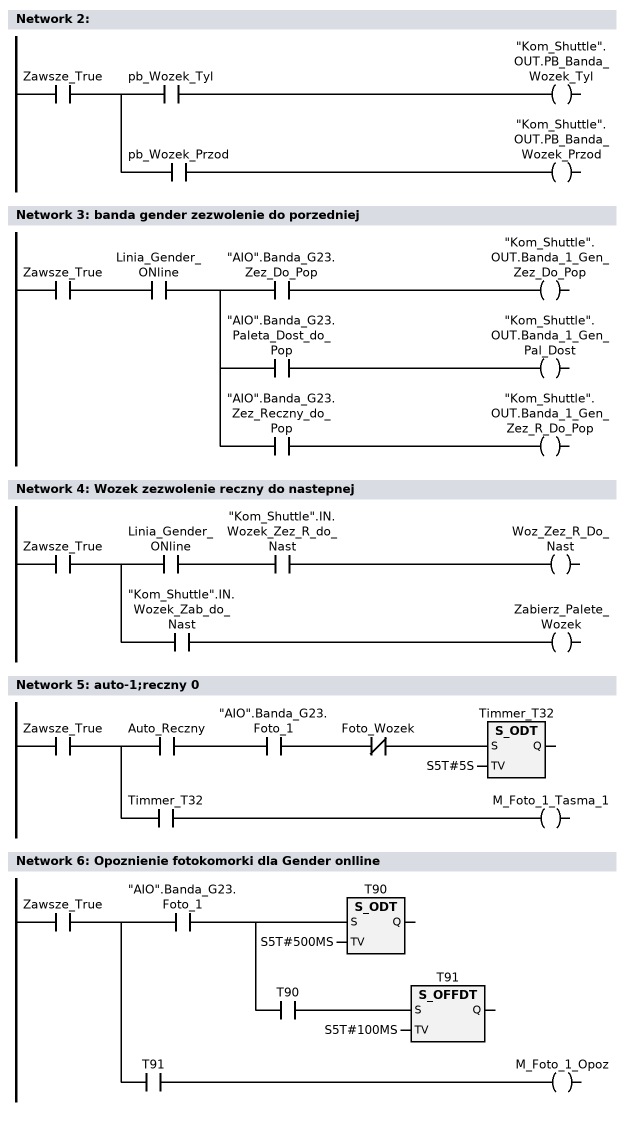
NETWORK
TITLE =
//Bity przychodzace od od bandy shuttle
      A     "Zawsze_True";
      =     L 1.0;
      A     L 1.0;
      A     "pb_Wozek_Tyl";
      =     "Kom_Shuttle".OUT.PB_Banda_Wozek_Tyl;
      A     L 1.0;
      A     "pb_Wozek_Przod";
      =     "Kom_Shuttle".OUT.PB_Banda_Wozek_Przod;
NETWORK
TITLE = banda gender zezwolenie do porzedniej
//Sygnal z poprzedniej
      A     "Zawsze_True";
      A     "Linia_Gender_ONline";
      =     L 1.0;
      A     L 1.0;
      A     "AIO".Banda_G23.Zez_Do_Pop;
      =     "Kom_Shuttle".OUT.Banda_1_Gen_Zez_Do_Pop;
      A     L 1.0;
      A     "AIO".Banda_G23.Paleta_Dost_do_Pop;
      =     "Kom_Shuttle".OUT.Banda_1_Gen_Pal_Dost;
      A     L 1.0;
      A     "AIO".Banda_G23.Zez_Reczny_do_Pop;
      =     "Kom_Shuttle".OUT.Banda_1_Gen_Zez_R_Do_Pop;
NETWORK
TITLE = Wozek zezwolenie reczny do nastepnej
      A     "Zawsze_True";
      =     L 1.0;
      A     L 1.0;
      A     "Linia_Gender_ONline";
      A     "Kom_Shuttle".IN.Wozek_Zez_R_do_Nast;
      =     "Woz_Zez_R_Do_Nast";
      A     L 1.0;
      A     "Kom_Shuttle".IN.Wozek_Zab_do_Nast;
      =     "Zabierz_Palete_Wozek";
NETWORK
TITLE = auto-1;reczny 0
//Opoznienie startu po polozeniu palety. Pomoc gdy paleta jest w strefie
      A     "Zawsze_True";
      =     L 1.0;
      A     L 1.0;
      A     "Auto_Reczny";
      A     "AIO".Banda_G23.Foto_1;
      AN    "Foto_Wozek";
      L     S5T#5S;
      SD    "Timmer_T32";
      NOP   0;
      NOP   0;
      NOP   0;
      NOP   0;
      A     L 1.0;
      A     "Timmer_T32";
      =     "M_Foto_1_Tasma_1";
NETWORK
TITLE = Opoznienie fotokomorki dla Gender onlline
      A     "Zawsze_True";
      =     L 1.0;
      A     L 1.0;
      A     "AIO".Banda_G23.Foto_1;
      =     L 1.1;
      A     L 1.1;
      L     S5T#500MS;
      SD    "T90";
      NOP   0;
      NOP   0;
      NOP   0;
      NOP   0;
      A     L 1.1;
      A     "T90";
      L     S5T#100MS;
      SF    "T91";
      NOP   0;
      NOP   0;
      NOP   0;
      NOP   0;
      A     L 1.0;
      A     "T91";
      =     "M_Foto_1_Opoz";
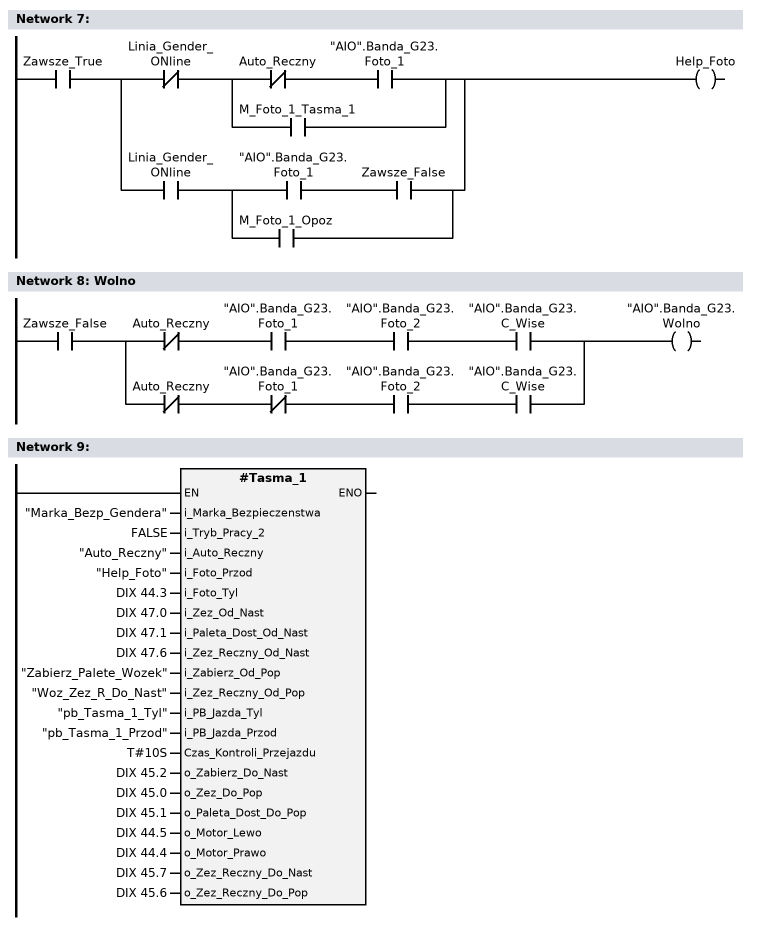
NETWORK
TITLE =
//Opoznienie wlotu bandy 1
      A     "Zawsze_True";
      A(;
      AN    "Linia_Gender_ONline";
      A(;
      AN    "Auto_Reczny";
      A     "AIO".Banda_G23.Foto_1;
      O     "M_Foto_1_Tasma_1";
      );
      O;
      A     "Linia_Gender_ONline";
      A(;
      A     "AIO".Banda_G23.Foto_1;
      A     "Zawsze_False";
      O     "M_Foto_1_Opoz";
      );
      );
      =     "Help_Foto";
NETWORK
TITLE = Wolno
////Silnik wolno  aby nie spadl z bandy
      A     "Zawsze_False";
      A(;
      AN    "Auto_Reczny";
      A     "AIO".Banda_G23.Foto_1;
      A     "AIO".Banda_G23.Foto_2;
      A     "AIO".Banda_G23.C_Wise;
      O;
      AN    "Auto_Reczny";
      AN    "AIO".Banda_G23.Foto_1;
      A     "AIO".Banda_G23.Foto_2;
      A     "AIO".Banda_G23.C_Wise;
      );
      =     "AIO".Banda_G23.Wolno;
NETWORK
TITLE =
//Tasma 1 adres 23
      CALL  #Tasma_1 (
           i_Marka_Bezpieczenstwa   := "Marka_Bezp_Gendera",
           i_Tryb_Pracy_2           := FALSE,
           i_Auto_Reczny            := "Auto_Reczny",
           i_Foto_Przod             := "Help_Foto",
           i_Foto_Tyl               := DIX 44.3,
           i_Zez_Od_Nast            := DIX 47.0,
           i_Paleta_Dost_Od_Nast    := DIX 47.1,
           i_Zez_Reczny_Od_Nast     := DIX 47.6,
           i_Zabierz_Od_Pop         := "Zabierz_Palete_Wozek",
           i_Zez_Reczny_Od_Pop      := "Woz_Zez_R_Do_Nast",
           i_PB_Jazda_Tyl           := "pb_Tasma_1_Tyl",
           i_PB_Jazda_Przod         := "pb_Tasma_1_Przod",
           Czas_Kontroli_Przejazdu  := T#10S,
           o_Zabierz_Do_Nast        := DIX 45.2,
           o_Zez_Do_Pop             := DIX 45.0,
           o_Paleta_Dost_Do_Pop     := DIX 45.1,
           o_Motor_Lewo             := DIX 44.5,
           o_Motor_Prawo            := DIX 44.4,
           o_Zez_Reczny_Do_Nast     := DIX 45.7,
           o_Zez_Reczny_Do_Pop      := DIX 45.6);	//kierunek normalny lini
      NOP   0;
NETWORK
TITLE =
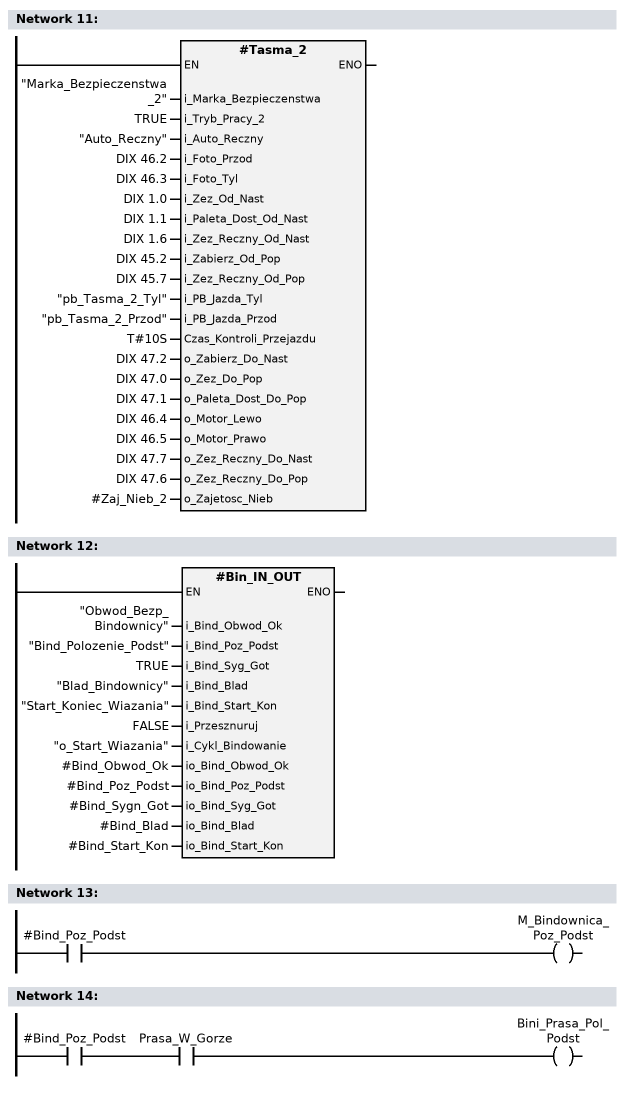
NETWORK
TITLE =
//Tasma 2 adres 24
      CALL  #Tasma_2 (
           i_Marka_Bezpieczenstwa   := "Marka_Bezpieczenstwa_2",
           i_Tryb_Pracy_2           := TRUE,
           i_Auto_Reczny            := "Auto_Reczny",
           i_Foto_Przod             := DIX 46.2,
           i_Foto_Tyl               := DIX 46.3,
           i_Zez_Od_Nast            := DIX 1.0,
           i_Paleta_Dost_Od_Nast    := DIX 1.1,
           i_Zez_Reczny_Od_Nast     := DIX 1.6,
           i_Zabierz_Od_Pop         := DIX 45.2,
           i_Zez_Reczny_Od_Pop      := DIX 45.7,
           i_PB_Jazda_Tyl           := "pb_Tasma_2_Tyl",
           i_PB_Jazda_Przod         := "pb_Tasma_2_Przod",
           Czas_Kontroli_Przejazdu  := T#10S,
           o_Zabierz_Do_Nast        := DIX 47.2,
           o_Zez_Do_Pop             := DIX 47.0,
           o_Paleta_Dost_Do_Pop     := DIX 47.1,
           o_Motor_Lewo             := DIX 46.4,
           o_Motor_Prawo            := DIX 46.5,
           o_Zez_Reczny_Do_Nast     := DIX 47.7,
           o_Zez_Reczny_Do_Pop      := DIX 47.6,
           o_Zajetosc_Nieb          := #Zaj_Nieb_2);	//kierunek normalny lini
      NOP   0;
NETWORK
TITLE =
//blok przejsciowy  do bindownicy
//(maskuje sygnal wejscia i wyjscia)
      CALL  #Bin_IN_OUT (
           i_Bind_Obwod_Ok          := "Obwod_Bezp_Bindownicy",
           i_Bind_Poz_Podst         := "Bind_Polozenie_Podst",
           i_Bind_Syg_Got           := TRUE,
           i_Bind_Blad              := "Blad_Bindownicy",
           i_Bind_Start_Kon         := "Start_Koniec_Wiazania",
           i_Przesznuruj            := FALSE,
           i_Cykl_Bindowanie        := "o_Start_Wiazania",
           io_Bind_Obwod_Ok         := #Bind_Obwod_Ok,
           io_Bind_Poz_Podst        := #Bind_Poz_Podst,
           io_Bind_Syg_Got          := #Bind_Sygn_Got,
           io_Bind_Blad             := #Bind_Blad,
           io_Bind_Start_Kon        := #Bind_Start_Kon);
NETWORK
TITLE =
      A     #Bind_Poz_Podst;
      =     "M_Bindownica_Poz_Podst";
NETWORK
TITLE =
      A     #Bind_Poz_Podst;
      A     "Prasa_W_Gorze";
      =     "Bini_Prasa_Pol_Podst";
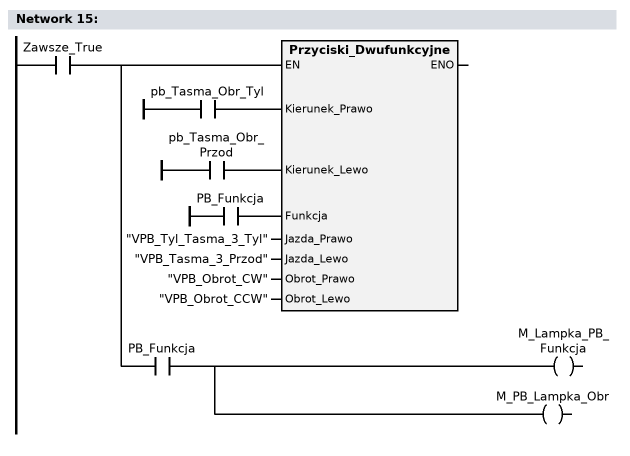
NETWORK
TITLE =
      A     "Zawsze_True";
      =     L 1.0;
      A     "pb_Tasma_Obr_Tyl";
      =     L 1.1;
      BLD   103;
      A     "pb_Tasma_Obr_Przod";
      =     L 1.2;
      BLD   103;
      A     "PB_Funkcja";
      =     L 1.3;
      BLD   103;
      A     L 1.0;
      JNB   _001;
      CALL  "Przyciski_Dwufunkcyjne" (
           Kierunek_Prawo           := L 1.1,
           Kierunek_Lewo            := L 1.2,
           Funkcja                  := L 1.3,
           Jazda_Prawo              := "VPB_Tyl_Tasma_3_Tyl",
           Jazda_Lewo               := "VPB_Tasma_3_Przod",
           Obrot_Prawo              := "VPB_Obrot_CW",
           Obrot_Lewo               := "VPB_Obrot_CCW");
_001: NOP   0;
      A     L 1.0;
      A     "PB_Funkcja";
      =     "M_Lampka_PB_Funkcja";
      =     "M_PB_Lampka_Obr";
NETWORK
TITLE =
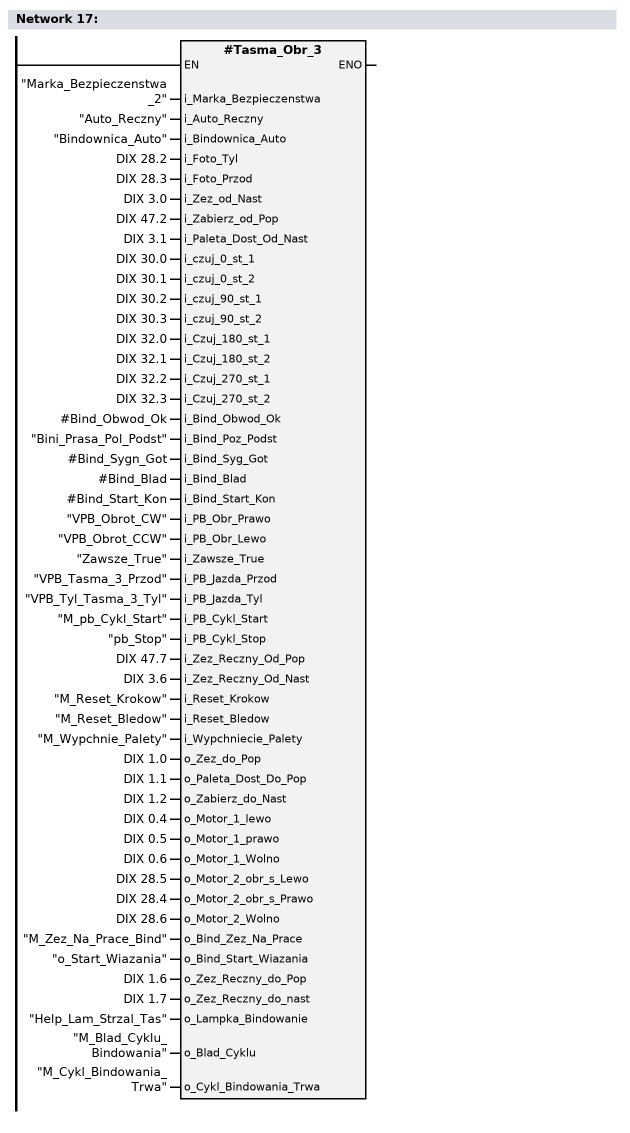
NETWORK
TITLE =
//bindownica z obrotnica
      CALL  #Tasma_Obr_3 (
           i_Marka_Bezpieczenstwa   := "Marka_Bezpieczenstwa_2",
           i_Auto_Reczny            := "Auto_Reczny",
           i_Bindownica_Auto        := "Bindownica_Auto",
           i_Foto_Tyl               := DIX 28.2,
           i_Foto_Przod             := DIX 28.3,
           i_Zez_od_Nast            := DIX 3.0,
           i_Zabierz_od_Pop         := DIX 47.2,
           i_Paleta_Dost_Od_Nast    := DIX 3.1,
           i_czuj_0_st_1            := DIX 30.0,
           i_czuj_0_st_2            := DIX 30.1,
           i_czuj_90_st_1           := DIX 30.2,
           i_czuj_90_st_2           := DIX 30.3,
           i_Czuj_180_st_1          := DIX 32.0,
           i_Czuj_180_st_2          := DIX 32.1,
           i_Czuj_270_st_1          := DIX 32.2,
           i_Czuj_270_st_2          := DIX 32.3,
           i_Bind_Obwod_Ok          := #Bind_Obwod_Ok,
           i_Bind_Poz_Podst         := "Bini_Prasa_Pol_Podst",
           i_Bind_Syg_Got           := #Bind_Sygn_Got,
           i_Bind_Blad              := #Bind_Blad,
           i_Bind_Start_Kon         := #Bind_Start_Kon,
           i_PB_Obr_Prawo           := "VPB_Obrot_CW",
           i_PB_Obr_Lewo            := "VPB_Obrot_CCW",
           i_Zawsze_True            := "Zawsze_True",
           i_PB_Jazda_Przod         := "VPB_Tasma_3_Przod",
           i_PB_Jazda_Tyl           := "VPB_Tyl_Tasma_3_Tyl",
           i_PB_Cykl_Start          := "M_pb_Cykl_Start",
           i_PB_Cykl_Stop           := "pb_Stop",
           i_Zez_Reczny_Od_Pop      := DIX 47.7,
           i_Zez_Reczny_Od_Nast     := DIX 3.6,
           i_Reset_Krokow           := "M_Reset_Krokow",
           i_Reset_Bledow           := "M_Reset_Bledow",
           i_Wypchniecie_Palety     := "M_Wypchnie_Palety",
           o_Zez_do_Pop             := DIX 1.0,
           o_Paleta_Dost_Do_Pop     := DIX 1.1,
           o_Zabierz_do_Nast        := DIX 1.2,
           o_Motor_1_lewo           := DIX 0.4,
           o_Motor_1_prawo          := DIX 0.5,
           o_Motor_1_Wolno          := DIX 0.6,
           o_Motor_2_obr_s_Lewo     := DIX 28.5,
           o_Motor_2_obr_s_Prawo    := DIX 28.4,
           o_Motor_2_Wolno          := DIX 28.6,
           o_Bind_Zez_Na_Prace      := "M_Zez_Na_Prace_Bind",
           o_Bind_Start_Wiazania    := "o_Start_Wiazania",
           o_Zez_Reczny_do_Pop      := DIX 1.6,
           o_Zez_Reczny_do_nast     := DIX 1.7,
           o_Lampka_Bindowanie      := "Help_Lam_Strzal_Tas",
           o_Blad_Cyklu             := "M_Blad_Cyklu_Bindowania",
           o_Cykl_Bindowania_Trwa   := "M_Cykl_Bindowania_Trwa");
NETWORK
TITLE = Zezwolenie na prase reczny
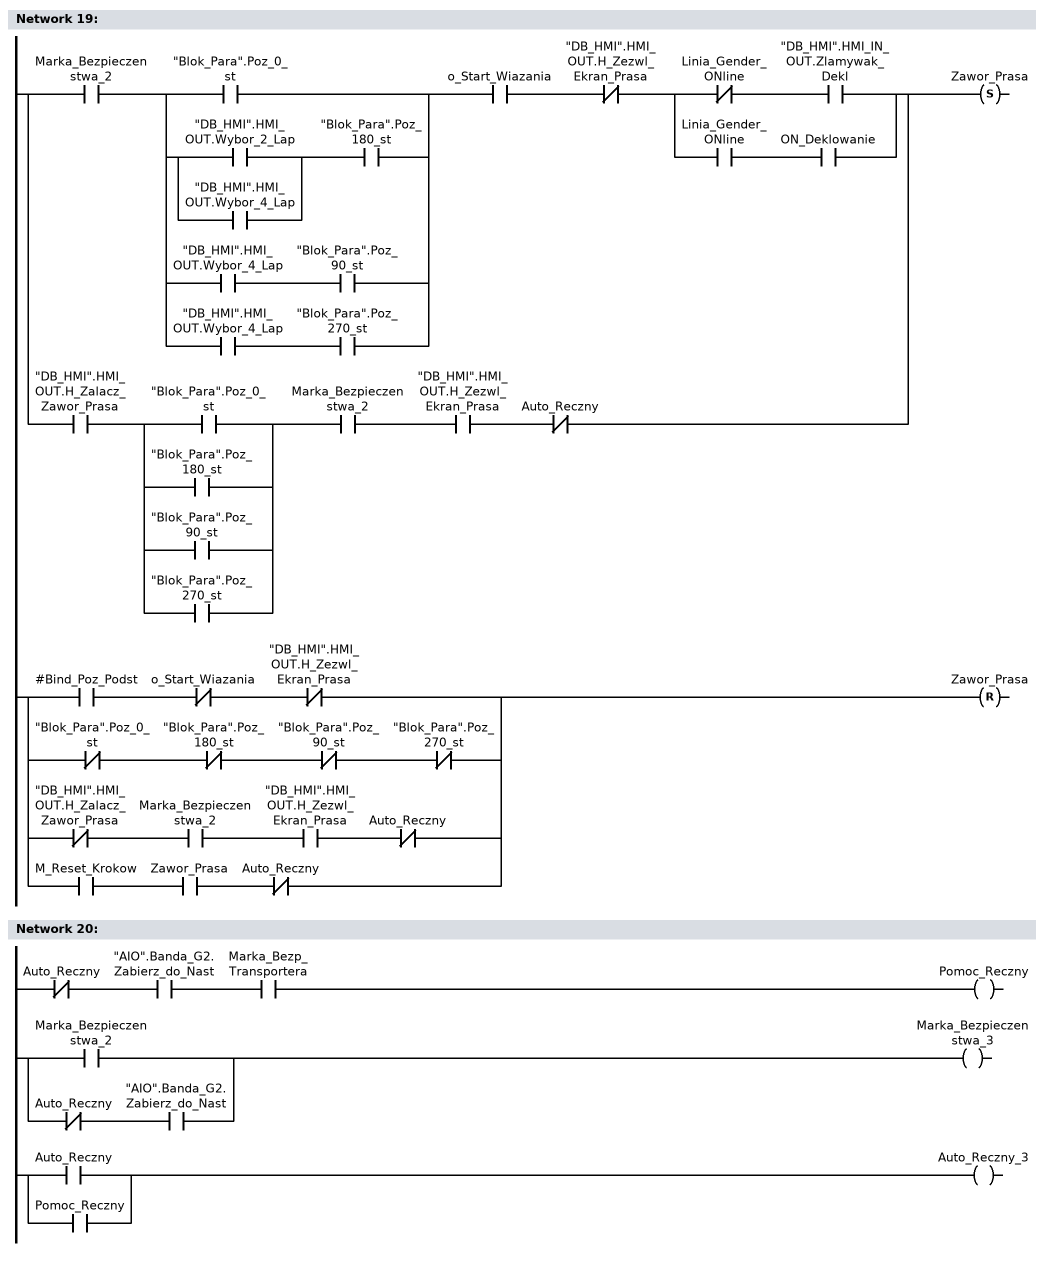
NETWORK
TITLE =
      A(;
      A     "Marka_Bezpieczenstwa_2";
      A(;
      O     "Blok_Para".Poz_0_st;
      O;
      A(;
      O     "DB_HMI".HMI_OUT.Wybor_2_Lap;
      O     "DB_HMI".HMI_OUT.Wybor_4_Lap;
      );
      A     "Blok_Para".Poz_180_st;
      O;
      A     "DB_HMI".HMI_OUT.Wybor_4_Lap;
      A     "Blok_Para".Poz_90_st;
      O;
      A     "DB_HMI".HMI_OUT.Wybor_4_Lap;
      A     "Blok_Para".Poz_270_st;
      );
      A     "o_Start_Wiazania";
      AN    "DB_HMI".HMI_OUT.H_Zezwl_Ekran_Prasa;
      A(;
      AN    "Linia_Gender_ONline";
      A     "DB_HMI".HMI_IN_OUT.Zlamywak_Dekl;
      O;
      A     "Linia_Gender_ONline";
      A     "ON_Deklowanie";
      );
      O;
      A     "DB_HMI".HMI_OUT.H_Zalacz_Zawor_Prasa;
      A(;
      O     "Blok_Para".Poz_0_st;
      O     "Blok_Para".Poz_180_st;
      O     "Blok_Para".Poz_90_st;
      O     "Blok_Para".Poz_270_st;
      );
      A     "Marka_Bezpieczenstwa_2";
      A     "DB_HMI".HMI_OUT.H_Zezwl_Ekran_Prasa;
      AN    "Auto_Reczny";
      );
      S     "Zawor_Prasa";
      A(;
      A     #Bind_Poz_Podst;
      AN    "o_Start_Wiazania";
      AN    "DB_HMI".HMI_OUT.H_Zezwl_Ekran_Prasa;
      O;
      AN    "Blok_Para".Poz_0_st;
      AN    "Blok_Para".Poz_180_st;
      AN    "Blok_Para".Poz_90_st;
      AN    "Blok_Para".Poz_270_st;
      O;
      AN    "DB_HMI".HMI_OUT.H_Zalacz_Zawor_Prasa;
      A     "Marka_Bezpieczenstwa_2";
      A     "DB_HMI".HMI_OUT.H_Zezwl_Ekran_Prasa;
      AN    "Auto_Reczny";
      O;
      A     "M_Reset_Krokow";
      A     "Zawor_Prasa";
      AN    "Auto_Reczny";
      );
      R     "Zawor_Prasa";
      NOP   0;
NETWORK
TITLE =
//Nowa Marka bepieczenstwa na wyjazd
//Marka bepieczenstwa przejsciowa
      AN    "Auto_Reczny";
      A     "AIO".Banda_G2.Zabierz_do_Nast;
      A     "Marka_Bezp_Transportera";
      =     "Pomoc_Reczny";
      A     "Marka_Bezpieczenstwa_2";
      O;
      AN    "Auto_Reczny";
      A     "AIO".Banda_G2.Zabierz_do_Nast;
      =     "Marka_Bezpieczenstwa_3";
//Jezeli marka bezpieczenstwa 3 auto zalaczone
      A     "Auto_Reczny";
      O;
      A     "Pomoc_Reczny";
      =     "Auto_Reczny_3";
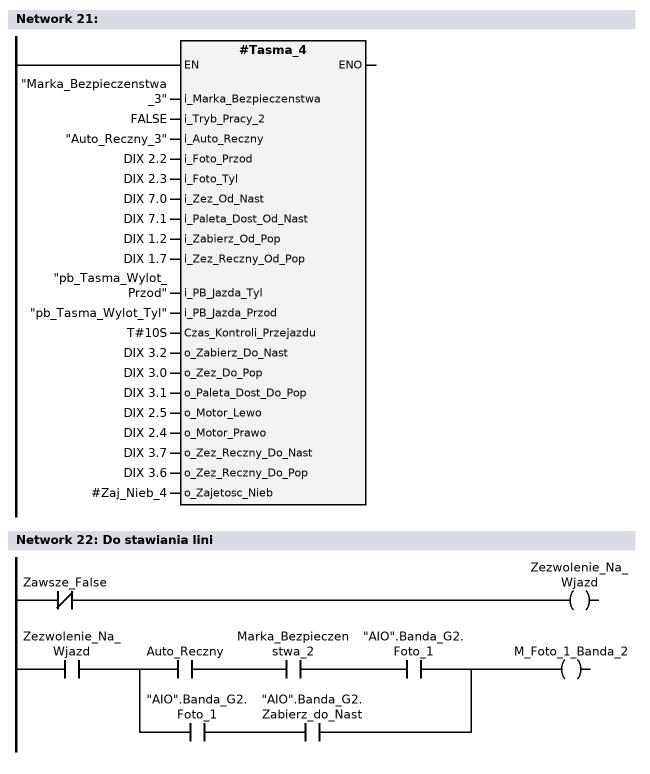
NETWORK
TITLE =
//Tasma 4 adres 2
//Ta tasma pod wzgledem bezpieczenstwa nalezy do lini i bindownicy
//Nastepna banda jest obrotnica
//
//
//
      CALL  #Tasma_4 (
           i_Marka_Bezpieczenstwa   := "Marka_Bezpieczenstwa_3",
           i_Tryb_Pracy_2           := FALSE,
           i_Auto_Reczny            := "Auto_Reczny_3",
           i_Foto_Przod             := DIX 2.2,
           i_Foto_Tyl               := DIX 2.3,
           i_Zez_Od_Nast            := DIX 7.0,
           i_Paleta_Dost_Od_Nast    := DIX 7.1,
           i_Zabierz_Od_Pop         := DIX 1.2,
           i_Zez_Reczny_Od_Pop      := DIX 1.7,
           i_PB_Jazda_Tyl           := "pb_Tasma_Wylot_Przod",
           i_PB_Jazda_Przod         := "pb_Tasma_Wylot_Tyl",
           Czas_Kontroli_Przejazdu  := T#10S,
           o_Zabierz_Do_Nast        := DIX 3.2,
           o_Zez_Do_Pop             := DIX 3.0,
           o_Paleta_Dost_Do_Pop     := DIX 3.1,
           o_Motor_Lewo             := DIX 2.5,
           o_Motor_Prawo            := DIX 2.4,
           o_Zez_Reczny_Do_Nast     := DIX 3.7,
           o_Zez_Reczny_Do_Pop      := DIX 3.6,
           o_Zajetosc_Nieb          := #Zaj_Nieb_4);	//kierunek normalny lini
NETWORK
TITLE = Do stawiania lini
//Banda 2. Uznawana za Wlot 1
//Uwaga By dzialolo nalezy wymusic true
      AN    "Zawsze_False";
      =     "Zezwolenie_Na_Wjazd";
//--
      A     "Zezwolenie_Na_Wjazd";
      A(;
      A     "Auto_Reczny";
      A     "Marka_Bezpieczenstwa_2";
      A     "AIO".Banda_G2.Foto_1;
      O;
      A     "AIO".Banda_G2.Foto_1;
      A     "AIO".Banda_G2.Zabierz_do_Nast;
      );
      =     "M_Foto_1_Banda_2";
END_FUNCTION_BLOCK

